KUKA KRL program: MyProgram_071().src

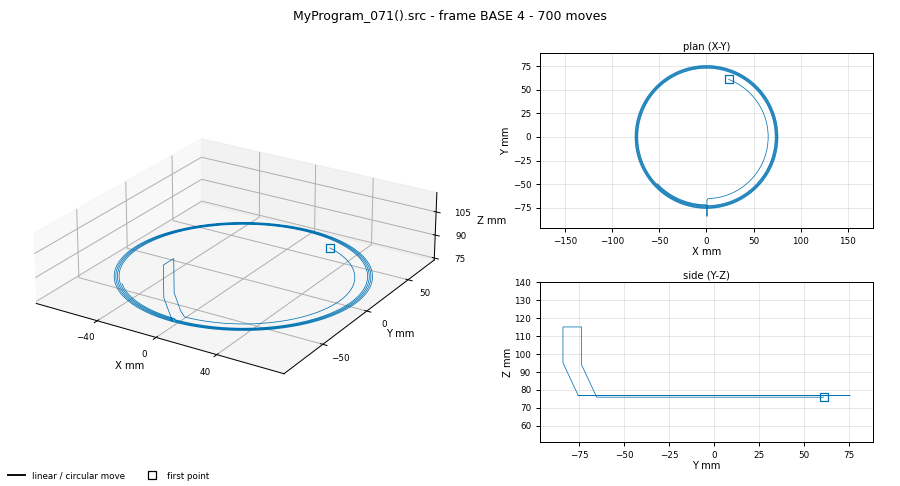
[picture p0: tool path of MyProgram_071().src in frame BASE 4, 700 of 700 moves have a stored position in this frame; points joined in program order, loops and branches not executed]
&ACCESS RVP
&REL 1
&PARAM TEMPLATE = C:\KRC\Roboter\Template\vorgabe
&PARAM EDITMASK = *
DEF MyProgram_071()
; ---- Setting reference (Base) ----
$BASE = BASE_DATA[4]

; --------------------------
; ---- Setting tool (TCP) ----
$TOOL = TOOL_DATA[3]
; --------------------------

$VEL.CP = VEL_APROX_PRINT
Startdeposition()
$VEL.CP = VEL_PRINT
LIN {X 23.5525,Y 61.0484,Z 76,A 61.9728,B 24.8705,C -2.6266,E1 25.0596,E2 22.1003} C_DIS
LIN {X 26.5205,Y 59.8189,Z 76,A 59.17,B 24.8707,C -2.6238,E1 25.0668,E2 24.903} C_DIS
LIN {X 29.4721,Y 58.4208,Z 76,A 56.3444,B 24.871,C -2.6212,E1 25.0738,E2 27.7274} C_DIS
LIN {X 32.2587,Y 56.9298,Z 76,A 53.5598,B 24.8714,C -2.617,E1 25.0807,E2 30.5137} C_DIS
LIN {X 35.0055,Y 55.2834,Z 76,A 50.8536,B 24.8716,C -2.6152,E1 25.0871,E2 33.2157} C_DIS
LIN {X 37.2904,Y 53.7671,Z 76,A 48.5544,B 24.8717,C -2.6139,E1 25.0924,E2 35.5104} C_DIS
LIN {X 39.6226,Y 52.0738,Z 76,A 45.8488,B 24.8726,C -2.6051,E1 25.0985,E2 38.2272} C_DIS
LIN {X 42.1324,Y 50.0649,Z 76,A 43.0554,B 24.873,C -2.6004,E1 25.1045,E2 41.021} C_DIS
LIN {X 44.5364,Y 47.9389,Z 76,A 40.2931,B 24.8735,C -2.596,E1 25.1102,E2 43.7826} C_DIS
LIN {X 46.2779,Y 46.26,Z 76,A 38.1504,B 24.874,C -2.591,E1 25.1145,E2 45.9282} C_DIS
LIN {X 48.4819,Y 43.9447,Z 76,A 35.3588,B 24.8745,C -2.585,E1 25.1198,E2 48.7216} C_DIS
LIN {X 50.5808,Y 41.5117,Z 76,A 32.55,B 24.8752,C -2.5787,E1 25.1249,E2 51.5324} C_DIS
LIN {X 52.564,Y 38.9698,Z 76,A 29.7557,B 24.8757,C -2.5727,E1 25.1296,E2 54.3278} C_DIS
LIN {X 54.4074,Y 36.352,Z 76,A 26.9662,B 24.8764,C -2.566,E1 25.134,E2 57.1193} C_DIS
LIN {X 55.9436,Y 33.9381,Z 76,A 24.5255,B 24.8769,C -2.5612,E1 25.1376,E2 59.559} C_DIS
LIN {X 57.326,Y 31.5494,Z 76,A 22.0724,B 24.8776,C -2.5539,E1 25.141,E2 62.0168} C_DIS
LIN {X 58.8026,Y 28.7034,Z 76,A 19.2702,B 24.8783,C -2.5463,E1 25.1445,E2 64.8219} C_DIS
LIN {X 60.1454,Y 25.7712,Z 76,A 16.4771,B 24.879,C -2.5392,E1 25.1477,E2 67.6166} C_DIS
LIN {X 61.3342,Y 22.7982,Z 76,A 13.8233,B 24.8794,C -2.5349,E1 25.1503,E2 70.2658} C_DIS
LIN {X 62.1448,Y 20.4847,Z 76,A 11.5626,B 24.8803,C -2.5257,E1 25.1524,E2 72.5355} C_DIS
LIN {X 63.0692,Y 17.4325,Z 76,A 8.7875,B 24.881,C -2.5178,E1 25.1545,E2 75.3133} C_DIS
LIN {X 63.8446,Y 14.3352,Z 76,A 6.0071,B 24.8818,C -2.5097,E1 25.1563,E2 78.0968} C_DIS
LIN {X 64.4679,Y 11.2033,Z 76,A 3.2328,B 24.8825,C -2.5017,E1 25.1577,E2 80.8738} C_DIS
LIN {X 64.9419,Y 8.0114,Z 76,A 0.4218,B 24.8833,C -2.4933,E1 25.1588,E2 83.6881} C_DIS
LIN {X 65.2564,Y 4.8203,Z 76,A -2.2442,B 24.8838,C -2.4881,E1 25.1595,E2 86.3505} C_DIS
LIN {X 65.39,Y 2.4055,Z 76,A -4.4684,B 24.8847,C -2.4787,E1 25.1597,E2 88.5837} C_DIS
LIN {X 65.4293,Y -0.8011,Z 76,A -7.1858,B 24.8853,C -2.4722,E1 25.1597,E2 91.3005} C_DIS
LIN {X 65.3532,Y -3.251,Z 76,A -9.4143,B 24.8861,C -2.4632,E1 25.1595,E2 93.5369} C_DIS
LIN {X 65.1176,Y -6.4286,Z 76,A -12.0528,B 24.8866,C -2.4583,E1 25.1588,E2 96.1713} C_DIS
LIN {X 64.8151,Y -8.9739,Z 76,A -14.3375,B 24.8873,C -2.4501,E1 25.158,E2 98.4619} C_DIS
LIN {X 64.3828,Y -11.6763,Z 76,A -16.6275,B 24.8878,C -2.4453,E1 25.157,E2 100.7497} C_DIS
LIN {X 63.8326,Y -14.3874,Z 76,A -19.1605,B 24.8887,C -2.4348,E1 25.1555,E2 103.2928} C_DIS
LIN {X 63.0604,Y -17.4644,Z 76,A -21.9235,B 24.8895,C -2.4265,E1 25.1535,E2 106.0594} C_DIS
LIN {X 62.242,Y -20.1845,Z 76,A -24.1704,B 24.8896,C -2.4251,E1 25.1516,E2 108.297} C_DIS
LIN {X 61.3315,Y -22.8052,Z 76,A -26.8132,B 24.8908,C -2.4121,E1 25.1491,E2 110.9556} C_DIS
LIN {X 60.2737,Y -25.4669,Z 76,A -29.2561,B 24.8913,C -2.4063,E1 25.1465,E2 113.3989} C_DIS
LIN {X 59.1341,Y -28.0135,Z 76,A -31.7276,B 24.8921,C -2.3983,E1 25.1436,E2 115.876} C_DIS
LIN {X 57.6977,Y -30.8641,Z 76,A -34.5052,B 24.8928,C -2.3906,E1 25.1401,E2 118.6571} C_DIS
LIN {X 56.1224,Y -33.6438,Z 76,A -37.287,B 24.8934,C -2.383,E1 25.1362,E2 121.4424} C_DIS
LIN {X 54.4127,Y -36.344,Z 76,A -40.0541,B 24.8941,C -2.376,E1 25.1319,E2 124.2122} C_DIS
LIN {X 52.4627,Y -39.1049,Z 76,A -42.9704,B 24.8947,C -2.3691,E1 25.1272,E2 127.1306} C_DIS
LIN {X 50.5595,Y -41.5372,Z 76,A -45.6811,B 24.8953,C -2.3619,E1 25.1224,E2 129.8458} C_DIS
LIN {X 48.5111,Y -43.9121,Z 76,A -48.3603,B 24.8958,C -2.3567,E1 25.1175,E2 132.5254} C_DIS
LIN {X 46.4255,Y -46.1105,Z 76,A -51.0603,B 24.8965,C -2.3491,E1 25.1122,E2 135.2318} C_DIS
LIN {X 44.1899,Y -48.2569,Z 76,A -53.7559,B 24.897,C -2.3432,E1 25.1067,E2 137.9302} C_DIS
LIN {X 41.9823,Y -50.1897,Z 76,A -56.2525,B 24.8973,C -2.3393,E1 25.1014,E2 140.4264} C_DIS
LIN {X 39.5895,Y -52.0987,Z 76,A -58.9906,B 24.898,C -2.3321,E1 25.0954,E2 143.1713} C_DIS
LIN {X 37.0025,Y -53.967,Z 76,A -61.7735,B 24.8984,C -2.3268,E1 25.089,E2 145.9571} C_DIS
LIN {X 34.3244,Y -55.7088,Z 76,A -64.5622,B 24.8989,C -2.3217,E1 25.0824,E2 148.7489} C_DIS
LIN {X 31.5458,Y -57.3279,Z 76,A -67.3726,B 24.8993,C -2.3169,E1 25.0756,E2 151.5623} C_DIS
LIN {X 28.694,Y -58.8072,Z 76,A -70.08,B 24.8995,C -2.3149,E1 25.0689,E2 154.2671} C_DIS
LIN {X 26.2021,Y -59.9577,Z 76,A -72.4647,B 24.8997,C -2.3117,E1 25.0628,E2 156.6533} C_DIS
LIN {X 23.7695,Y -60.9632,Z 76,A -74.8521,B 24.9002,C -2.3065,E1 25.0566,E2 159.0477} C_DIS
LIN {X 20.8144,Y -62.0342,Z 76,A -77.6031,B 24.9005,C -2.3031,E1 25.0493,E2 161.8014} C_DIS
LIN {X 17.8967,Y -62.938,Z 76,A -80.1335,B 24.9005,C -2.3035,E1 25.0426,E2 164.3262} C_DIS
LIN {X 15.2789,Y -63.6246,Z 76,A -82.6105,B 24.9009,C -2.2986,E1 25.0358,E2 166.8112} C_DIS
LIN {X 12.3023,Y -64.2661,Z 76,A -85.3165,B 24.9011,C -2.2954,E1 25.0284,E2 169.5215} C_DIS
LIN {X 10.0745,Y -64.6528,Z 76,A -87.1823,B 24.9011,C -2.2966,E1 25.0233,E2 171.3825} C_DIS
LIN {X 7.1628,Y -65.0407,Z 76,A -89.7299,B 24.9011,C -2.2956,E1 25.0162,E2 173.9306} C_DIS
LIN {X 4.6112,Y -65.2706,Z 76,A -91.976,B 24.9012,C -2.2945,E1 25.01,E2 176.1783} C_DIS
LIN {X 1.6014,Y -65.4146,Z 76,A -94.7265,B 24.9015,C -2.2909,E1 25.0023,E2 178.9364} C_DIS
LIN {X 1.6014,Y -65.4146,Z 76,A -94.7265,B 24.9015,C -2.2909,E1 25.0023,E2 178.9364} C_DIS
Enddeposition()
LIN {X 0.4347,Y -67.5421,Z 80.5315,A -94.7713,B 24.8999,C -2.3098,E1 25.0023,E2 178.9364} C_DIS
LIN {X 0.5123,Y -73.8809,Z 94.1262,A -94.7477,B 24.9008,C -2.2999,E1 25.0023,E2 178.9364} C_DIS
LIN {X 0.5123,Y -73.8809,Z 115.1262,A -95.1061,B 24.8873,C -2.4507,E1 25.0023,E2 178.9364} C_DIS
LIN {X 0.5071,Y -84.2101,Z 115.1262,A -95.3701,B 24.9039,C -2.2639,E1 25.0003,E2 179.6442} C_DIS
LIN {X 0.5071,Y -84.2101,Z 95.1262,A -95.0293,B 24.9157,C -2.1203,E1 25.0003,E2 179.6442} C_DIS
LIN {X 0.5079,Y -77.8709,Z 81.5315,A -95.0515,B 24.9149,C -2.1297,E1 25.0003,E2 179.6442} C_DIS
LIN {X 0.5081,Y -75.7578,Z 77,A -95.0604,B 24.9146,C -2.1334,E1 25.0003,E2 179.6442} C_DIS
Startdeposition()
$VEL.CP = VEL_PRINT
LIN {X -1.8593,Y -75.7398,Z 77,A -96.8129,B 24.9146,C -2.1341,E1 24.9954,E2 181.3953} C_DIS
LIN {X -4.4218,Y -75.6324,Z 77,A -98.7832,B 24.9146,C -2.1331,E1 24.9899,E2 183.3684} C_DIS
LIN {X -7.315,Y -75.4081,Z 77,A -100.9558,B 24.9146,C -2.1338,E1 24.9839,E2 185.5404} C_DIS
LIN {X -9.1634,Y -75.2058,Z 77,A -102.3625,B 24.9146,C -2.1339,E1 24.98,E2 186.9476} C_DIS
LIN {X -11.0062,Y -74.9583,Z 77,A -103.7692,B 24.9146,C -2.1342,E1 24.9761,E2 188.3547} C_DIS
LIN {X -12.8425,Y -74.6656,Z 77,A -105.1758,B 24.9146,C -2.1346,E1 24.9722,E2 189.7617} C_DIS
LIN {X -14.671,Y -74.328,Z 77,A -106.5836,B 24.9146,C -2.1351,E1 24.9683,E2 191.1699} C_DIS
LIN {X -16.4907,Y -73.9455,Z 77,A -107.9913,B 24.9145,C -2.1357,E1 24.9645,E2 192.5779} C_DIS
LIN {X -18.3004,Y -73.5185,Z 77,A -109.3994,B 24.9144,C -2.1364,E1 24.9607,E2 193.9863} C_DIS
LIN {X -20.0992,Y -73.0473,Z 77,A -110.8076,B 24.9144,C -2.1372,E1 24.9569,E2 195.3947} C_DIS
LIN {X -22.3492,Y -72.3898,Z 77,A -112.7026,B 24.9144,C -2.1352,E1 24.9518,E2 197.2976} C_DIS
LIN {X -24.6464,Y -71.6417,Z 77,A -114.4045,B 24.9141,C -2.1399,E1 24.9473,E2 198.9916} C_DIS
LIN {X -26.595,Y -70.9403,Z 77,A -116.1762,B 24.9144,C -2.136,E1 24.9426,E2 200.7762} C_DIS
LIN {X -28.8898,Y -70.0376,Z 77,A -117.9878,B 24.9142,C -2.1392,E1 24.9379,E2 202.5843} C_DIS
LIN {X -31.4481,Y -68.9268,Z 77,A -119.9663,B 24.9137,C -2.1448,E1 24.9329,E2 204.5541} C_DIS
LIN {X -33.8074,Y -67.8001,Z 77,A -121.9882,B 24.9137,C -2.146,E1 24.9278,E2 206.5783} C_DIS
LIN {X -35.7143,Y -66.8167,Z 77,A -123.8482,B 24.9139,C -2.142,E1 24.9232,E2 208.453} C_DIS
LIN {X -38.0527,Y -65.5124,Z 77,A -125.5985,B 24.9132,C -2.1518,E1 24.919,E2 210.1852} C_DIS
LIN {X -39.7443,Y -64.5009,Z 77,A -127.2084,B 24.9132,C -2.1509,E1 24.9151,E2 211.8022} C_DIS
LIN {X -41.9983,Y -63.0557,Z 77,A -129.1259,B 24.9128,C -2.1567,E1 24.9106,E2 213.712} C_DIS
LIN {X -43.5988,Y -61.9604,Z 77,A -130.5959,B 24.9126,C -2.159,E1 24.9073,E2 215.1815} C_DIS
LIN {X -45.1317,Y -60.8531,Z 77,A -132.0335,B 24.9124,C -2.1613,E1 24.904,E2 216.6189} C_DIS
LIN {X -46.6116,Y -59.7272,Z 77,A -133.4456,B 24.9122,C -2.1636,E1 24.9009,E2 218.0305} C_DIS
LIN {X -48.6075,Y -58.1131,Z 77,A -135.4115,B 24.912,C -2.1666,E1 24.8967,E2 219.9968} C_DIS
LIN {X -50.1864,Y -56.7565,Z 77,A -136.9756,B 24.9117,C -2.1698,E1 24.8934,E2 221.5594} C_DIS
LIN {X -51.5641,Y -55.5078,Z 77,A -138.3881,B 24.9115,C -2.1724,E1 24.8905,E2 222.9712} C_DIS
LIN {X -53.4929,Y -53.6507,Z 77,A -140.431,B 24.9112,C -2.1762,E1 24.8864,E2 225.0138} C_DIS
LIN {X -54.8709,Y -52.2414,Z 77,A -141.9205,B 24.9109,C -2.1794,E1 24.8835,E2 226.5022} C_DIS
LIN {X -56.6821,Y -50.2695,Z 77,A -143.9552,B 24.9106,C -2.1836,E1 24.8797,E2 228.5358} C_DIS
LIN {X -57.9711,Y -48.7784,Z 77,A -145.4534,B 24.9103,C -2.1868,E1 24.877,E2 230.0333} C_DIS
LIN {X -59.1507,Y -47.341,Z 77,A -147.109,B 24.9105,C -2.184,E1 24.874,E2 231.7032} C_DIS
LIN {X -60.8531,Y -45.1317,Z 77,A -148.9877,B 24.9097,C -2.1946,E1 24.8709,E2 233.5655} C_DIS
LIN {X -61.9424,Y -43.6247,Z 77,A -150.4018,B 24.9094,C -2.1979,E1 24.8686,E2 234.9788} C_DIS
LIN {X -62.9943,Y -42.0915,Z 77,A -151.8158,B 24.9091,C -2.2012,E1 24.8664,E2 236.3918} C_DIS
LIN {X -64.1223,Y -40.3503,Z 77,A -153.595,B 24.9091,C -2.2002,E1 24.8637,E2 238.1825} C_DIS
LIN {X -65.5927,Y -37.9129,Z 77,A -155.7542,B 24.9087,C -2.2057,E1 24.8606,E2 240.3398} C_DIS
LIN {X -66.9995,Y -35.3671,Z 77,A -157.8935,B 24.9081,C -2.213,E1 24.8578,E2 242.4728} C_DIS
LIN {X -68.0859,Y -33.2307,Z 77,A -159.8507,B 24.9081,C -2.2145,E1 24.8554,E2 244.437} C_DIS
LIN {X -69.2629,Y -30.7021,Z 77,A -161.7188,B 24.907,C -2.2262,E1 24.8532,E2 246.2875} C_DIS
LIN {X -69.9955,Y -28.9931,Z 77,A -163.1343,B 24.9067,C -2.2299,E1 24.8517,E2 247.7019} C_DIS
LIN {X -70.686,Y -27.2666,Z 77,A -164.5499,B 24.9064,C -2.2338,E1 24.8502,E2 249.1163} C_DIS
LIN {X -71.3338,Y -25.5237,Z 77,A -165.9652,B 24.9061,C -2.2376,E1 24.8489,E2 250.5303} C_DIS
LIN {X -71.9031,Y -23.8711,Z 77,A -167.3043,B 24.9058,C -2.2411,E1 24.8477,E2 251.8687} C_DIS
LIN {X -72.733,Y -21.2083,Z 77,A -169.4276,B 24.9053,C -2.2471,E1 24.846,E2 253.99} C_DIS
LIN {X -73.4125,Y -18.7184,Z 77,A -171.4427,B 24.9049,C -2.2514,E1 24.8445,E2 256.0064} C_DIS
LIN {X -73.9744,Y -16.3584,Z 77,A -173.4176,B 24.9047,C -2.2537,E1 24.8433,E2 257.9874} C_DIS
LIN {X -74.4826,Y -13.8676,Z 77,A -175.2484,B 24.904,C -2.2618,E1 24.8423,E2 259.8099} C_DIS
LIN {X -74.9256,Y -11.2269,Z 77,A -177.2155,B 24.9034,C -2.2694,E1 24.8414,E2 261.7704} C_DIS
LIN {X -75.246,Y -8.8201,Z 77,A -179.1504,B 24.9031,C -2.2728,E1 24.8407,E2 263.7087} C_DIS
LIN {X -75.4833,Y -6.5002,Z 77,A 179.168,B 24.9024,C -2.2803,E1 24.8403,E2 265.3827} C_DIS
LIN {X -75.6652,Y -3.8289,Z 77,A 177.1202,B 24.9019,C -2.2861,E1 24.8399,E2 267.4288} C_DIS
LIN {X -75.7549,Y -1.0413,Z 77,A 174.7529,B 24.9019,C -2.2868,E1 24.8398,E2 269.8088} C_DIS
LIN {X -75.7398,Y 1.8593,Z 77,A 172.7949,B 24.9008,C -2.2992,E1 24.8398,E2 271.7488} C_DIS
LIN {X -75.6761,Y 3.606,Z 77,A 171.3838,B 24.9006,C -2.3014,E1 24.84,E2 273.1633} C_DIS
LIN {X -75.4937,Y 6.3697,Z 77,A 169.3521,B 24.8999,C -2.3095,E1 24.8404,E2 275.1878} C_DIS
LIN {X -75.301,Y 8.3507,Z 77,A 167.8383,B 24.8995,C -2.3141,E1 24.8409,E2 276.6998} C_DIS
LIN {X -75.0734,Y 10.1962,Z 77,A 166.4219,B 24.8992,C -2.3183,E1 24.8414,E2 278.1146} C_DIS
LIN {X -74.7112,Y 12.5698,Z 77,A 164.3699,B 24.8992,C -2.3185,E1 24.8423,E2 280.1781} C_DIS
LIN {X -74.1199,Y 15.6913,Z 77,A 162.1728,B 24.8981,C -2.3309,E1 24.8435,E2 282.3588} C_DIS
LIN {X -73.7125,Y 17.5056,Z 77,A 160.7567,B 24.8977,C -2.3351,E1 24.8444,E2 283.7732} C_DIS
LIN {X -73.2607,Y 19.3093,Z 77,A 159.3407,B 24.8973,C -2.3392,E1 24.8453,E2 285.1875} C_DIS
LIN {X -72.7647,Y 21.1014,Z 77,A 157.9247,B 24.897,C -2.3434,E1 24.8464,E2 286.6018} C_DIS
LIN {X -72.225,Y 22.8808,Z 77,A 156.5087,B 24.8966,C -2.3475,E1 24.8476,E2 288.0161} C_DIS
LIN {X -71.6417,Y 24.6464,Z 77,A 154.8804,B 24.8966,C -2.3466,E1 24.8491,E2 289.6558} C_DIS
LIN {X -70.7255,Y 27.1623,Z 77,A 153.045,B 24.8957,C -2.3572,E1 24.8508,E2 291.4763} C_DIS
LIN {X -69.7451,Y 29.5874,Z 77,A 151.0139,B 24.8953,C -2.3619,E1 24.853,E2 293.5074} C_DIS
LIN {X -68.9268,Y 31.4481,Z 77,A 149.3728,B 24.8951,C -2.3641,E1 24.8549,E2 295.1524} C_DIS
LIN {X -67.7226,Y 33.9638,Z 77,A 147.3824,B 24.8943,C -2.3731,E1 24.8573,E2 297.1321} C_DIS
LIN {X -66.8686,Y 35.6155,Z 77,A 145.967,B 24.894,C -2.3769,E1 24.8591,E2 298.5458} C_DIS
LIN {X -65.7568,Y 37.6275,Z 77,A 144.0566,B 24.8939,C -2.3779,E1 24.8617,E2 300.464} C_DIS
LIN {X -64.5009,Y 39.7443,Z 77,A 142.3527,B 24.8931,C -2.3868,E1 24.8642,E2 302.1553} C_DIS
LIN {X -62.9943,Y 42.0915,Z 77,A 140.23,B 24.8926,C -2.3923,E1 24.8674,E2 304.2755} C_DIS
LIN {X -61.6349,Y 44.0557,Z 77,A 138.1767,B 24.8926,C -2.3914,E1 24.8707,E2 306.3411} C_DIS
LIN {X -59.7272,Y 46.6116,Z 77,A 135.9861,B 24.8916,C -2.403,E1 24.8744,E2 308.5144} C_DIS
LIN {X -58.0424,Y 48.6926,Z 77,A 133.9493,B 24.8912,C -2.408,E1 24.878,E2 310.5489} C_DIS
LIN {X -56.8299,Y 50.1023,Z 77,A 132.5264,B 24.8909,C -2.4111,E1 24.8806,E2 311.9707} C_DIS
LIN {X -55.5078,Y 51.5641,Z 77,A 130.7939,B 24.8911,C -2.409,E1 24.8839,E2 313.7159} C_DIS
LIN {X -53.5723,Y 53.5723,Z 77,A 128.6328,B 24.8907,C -2.4128,E1 24.8881,E2 315.8771} C_DIS
LIN {X -51.3931,Y 55.6647,Z 77,A 126.4255,B 24.8901,C -2.42,E1 24.8926,E2 318.0763} C_DIS
LIN {X -49.5701,Y 57.2947,Z 77,A 124.7509,B 24.8893,C -2.4283,E1 24.8961,E2 319.7376} C_DIS
LIN {X -47.4277,Y 59.0805,Z 77,A 122.4512,B 24.8893,C -2.4283,E1 24.9011,E2 322.0462} C_DIS
LIN {X -45.1317,Y 60.8531,Z 77,A 120.4362,B 24.8885,C -2.4372,E1 24.9055,E2 324.0472} C_DIS
LIN {X -43.6247,Y 61.9424,Z 77,A 119.0235,B 24.8883,C -2.4398,E1 24.9087,E2 325.4585} C_DIS
LIN {X -42.0915,Y 62.9943,Z 77,A 117.611,B 24.888,C -2.4424,E1 24.912,E2 326.8696} C_DIS
LIN {X -40.6267,Y 63.9481,Z 77,A 116.0362,B 24.8884,C -2.4387,E1 24.9157,E2 328.4583} C_DIS
LIN {X -38.1494,Y 65.4568,Z 77,A 114.0099,B 24.8876,C -2.4467,E1 24.9206,E2 330.4716} C_DIS
LIN {X -35.8471,Y 66.7446,Z 77,A 112.074,B 24.8872,C -2.4516,E1 24.9253,E2 332.4015} C_DIS
LIN {X -34.1631,Y 67.6222,Z 77,A 110.6284,B 24.887,C -2.4537,E1 24.9289,E2 333.846} C_DIS
LIN {X -32.4932,Y 68.4403,Z 77,A 109.0424,B 24.8872,C -2.4514,E1 24.9329,E2 335.4415} C_DIS
LIN {X -29.9521,Y 69.5899,Z 77,A 107.101,B 24.8865,C -2.4587,E1 24.9378,E2 337.3703} C_DIS
LIN {X -28.132,Y 70.3461,Z 77,A 105.614,B 24.8863,C -2.4608,E1 24.9416,E2 338.8555} C_DIS
LIN {X -26.3971,Y 71.0153,Z 77,A 103.9456,B 24.8868,C -2.456,E1 24.946,E2 340.5387} C_DIS
LIN {X -23.8711,Y 71.9031,Z 77,A 102.1647,B 24.886,C -2.4647,E1 24.9507,E2 342.3025} C_DIS
LIN {X -21.2083,Y 72.733,Z 77,A 100.0588,B 24.8858,C -2.4671,E1 24.9563,E2 344.4062} C_DIS
LIN {X -19.3093,Y 73.2607,Z 77,A 98.565,B 24.8856,C -2.4685,E1 24.9603,E2 345.899} C_DIS
LIN {X -17.5056,Y 73.7125,Z 77,A 97.1554,B 24.8856,C -2.4697,E1 24.9642,E2 347.3076} C_DIS
LIN {X -15.6913,Y 74.1199,Z 77,A 95.4735,B 24.8861,C -2.4639,E1 24.9688,E2 349.0054} C_DIS
LIN {X -13.0623,Y 74.6275,Z 77,A 93.7096,B 24.8853,C -2.4722,E1 24.9736,E2 350.7516} C_DIS
LIN {X -10.8615,Y 74.9789,Z 77,A 91.8499,B 24.8856,C -2.4688,E1 24.9788,E2 352.6208} C_DIS
LIN {X -8.3507,Y 75.301,Z 77,A 89.909,B 24.8856,C -2.4692,E1 24.9841,E2 354.5621} C_DIS
LIN {X -5.5734,Y 75.5573,Z 77,A 88.0013,B 24.885,C -2.4754,E1 24.9894,E2 356.456} C_DIS
LIN {X -2.9846,Y 75.7029,Z 77,A 86.0273,B 24.885,C -2.4758,E1 24.9949,E2 358.4296} C_DIS
LIN {X -1.0663,Y 75.7544,Z 77,A 84.3242,B 24.8855,C -2.4695,E1 24.9997,E2 360.1476} C_DIS
LIN {X 1.8593,Y 75.7398,Z 77,A 82.3732,B 24.8849,C -2.4767,E1 25.0051,E2 362.0813} C_DIS
LIN {X 3.606,Y 75.6761,Z 77,A 81.0424,B 24.8849,C -2.4766,E1 25.0088,E2 363.412} C_DIS
LIN {X 5.5734,Y 75.5573,Z 77,A 79.5609,B 24.8849,C -2.4768,E1 25.0129,E2 364.8924} C_DIS
LIN {X 8.3507,Y 75.301,Z 77,A 77.4522,B 24.8849,C -2.4766,E1 25.0188,E2 367.0003} C_DIS
LIN {X 10.4168,Y 75.042,Z 77,A 75.6607,B 24.8855,C -2.4704,E1 25.0238,E2 368.8049} C_DIS
LIN {X 12.8425,Y 74.6656,Z 77,A 74.0143,B 24.885,C -2.4755,E1 25.0283,E2 370.4376} C_DIS
LIN {X 14.671,Y 74.328,Z 77,A 72.6093,B 24.885,C -2.4749,E1 25.0322,E2 371.8423} C_DIS
LIN {X 17.2224,Y 73.7779,Z 77,A 70.6125,B 24.8852,C -2.4733,E1 25.0376,E2 373.8403} C_DIS
LIN {X 19.2371,Y 73.2792,Z 77,A 69.0808,B 24.8852,C -2.4734,E1 25.0417,E2 375.3695} C_DIS
LIN {X 21.1014,Y 72.7647,Z 77,A 67.5473,B 24.8854,C -2.4705,E1 25.0459,E2 376.9073} C_DIS
LIN {X 23.6061,Y 71.9903,Z 77,A 65.6202,B 24.8854,C -2.4705,E1 25.051,E2 378.8309} C_DIS
LIN {X 25.4184,Y 71.3708,Z 77,A 64.1842,B 24.8855,C -2.4696,E1 25.0548,E2 380.2662} C_DIS
LIN {X 27.2297,Y 70.6999,Z 77,A 62.7376,B 24.8856,C -2.4686,E1 25.0586,E2 381.712} C_DIS
LIN {X 28.8898,Y 70.0376,Z 77,A 61.378,B 24.8858,C -2.467,E1 25.0621,E2 383.0723} C_DIS
LIN {X 30.6872,Y 69.2694,Z 77,A 59.9134,B 24.8858,C -2.4658,E1 25.0658,E2 384.5362} C_DIS
LIN {X 32.3927,Y 68.4886,Z 77,A 58.497,B 24.886,C -2.4642,E1 25.0694,E2 385.9528} C_DIS
LIN {X 34.5281,Y 67.4357,Z 77,A 56.6311,B 24.8864,C -2.4602,E1 25.0741,E2 387.8232} C_DIS
LIN {X 36.5315,Y 66.3734,Z 77,A 54.7344,B 24.8871,C -2.4528,E1 25.0788,E2 389.732} C_DIS
LIN {X 38.8537,Y 65.0405,Z 77,A 52.9638,B 24.8867,C -2.457,E1 25.083,E2 391.4871} C_DIS
LIN {X 41.2163,Y 63.5696,Z 77,A 50.8746,B 24.887,C -2.4542,E1 25.0879,E2 393.5762} C_DIS
LIN {X 42.769,Y 62.5356,Z 77,A 49.4693,B 24.8871,C -2.4521,E1 25.0912,E2 394.9818} C_DIS
LIN {X 44.2908,Y 61.4672,Z 77,A 48.0597,B 24.8874,C -2.4497,E1 25.0944,E2 396.3923} C_DIS
LIN {X 45.8751,Y 60.2947,Z 77,A 46.5836,B 24.8876,C -2.4475,E1 25.0977,E2 397.8683} C_DIS
LIN {X 47.341,Y 59.1507,Z 77,A 45.183,B 24.8878,C -2.4451,E1 25.1008,E2 399.2693} C_DIS
LIN {X 49.3944,Y 57.4462,Z 77,A 43.1632,B 24.8882,C -2.4412,E1 25.1051,E2 401.2904} C_DIS
LIN {X 50.796,Y 56.2108,Z 77,A 41.7578,B 24.8884,C -2.4387,E1 25.108,E2 402.6963} C_DIS
LIN {X 52.2414,Y 54.8709,Z 77,A 40.2824,B 24.8886,C -2.4361,E1 25.111,E2 404.1718} C_DIS
LIN {X 53.4929,Y 53.6507,Z 77,A 38.9583,B 24.8889,C -2.4332,E1 25.1137,E2 405.497} C_DIS
LIN {X 54.7934,Y 52.3217,Z 77,A 37.5588,B 24.8891,C -2.4304,E1 25.1164,E2 406.8971} C_DIS
LIN {X 56.1364,Y 50.8791,Z 77,A 36.0839,B 24.8894,C -2.4276,E1 25.1192,E2 408.3723} C_DIS
LIN {X 57.3681,Y 49.4861,Z 77,A 34.6847,B 24.8897,C -2.4246,E1 25.1217,E2 409.7722} C_DIS
LIN {X 58.5653,Y 48.0633,Z 77,A 33.2856,B 24.89,C -2.4216,E1 25.1242,E2 411.1721} C_DIS
LIN {X 59.7272,Y 46.6116,Z 77,A 31.8867,B 24.8902,C -2.4185,E1 25.1267,E2 412.5718} C_DIS
LIN {X 60.8531,Y 45.1317,Z 77,A 30.4882,B 24.8905,C -2.4153,E1 25.129,E2 413.9712} C_DIS
LIN {X 61.8776,Y 43.7155,Z 77,A 29.0846,B 24.891,C -2.4096,E1 25.1313,E2 415.3813} C_DIS
LIN {X 63.4447,Y 41.4084,Z 77,A 27.0673,B 24.8913,C -2.407,E1 25.1344,E2 417.3947} C_DIS
LIN {X 64.7248,Y 39.3758,Z 77,A 25.1661,B 24.8919,C -2.3998,E1 25.1372,E2 419.3033} C_DIS
LIN {X 65.8645,Y 37.44,Z 77,A 23.3912,B 24.8925,C -2.3931,E1 25.1397,E2 421.0849} C_DIS
LIN {X 67.2499,Y 34.8916,Z 77,A 21.4001,B 24.8925,C -2.3931,E1 25.1423,E2 423.0655} C_DIS
LIN {X 68.0859,Y 33.2307,Z 77,A 19.8587,B 24.8932,C -2.3852,E1 25.1442,E2 424.6174} C_DIS
LIN {X 69.2629,Y 30.7021,Z 77,A 17.9065,B 24.8934,C -2.384,E1 25.1465,E2 426.5619} C_DIS
LIN {X 70.3461,Y 28.132,Z 77,A 15.8104,B 24.8939,C -2.3783,E1 25.1487,E2 428.6598} C_DIS
LIN {X 71.0153,Y 26.3971,Z 77,A 14.3101,B 24.8945,C -2.3714,E1 25.1502,E2 430.168} C_DIS
LIN {X 71.9031,Y 23.8711,Z 77,A 12.3926,B 24.8947,C -2.3687,E1 25.152,E2 432.0811} C_DIS
LIN {X 72.6863,Y 21.3657,Z 77,A 10.4001,B 24.8953,C -2.3626,E1 25.1536,E2 434.0768} C_DIS
LIN {X 73.3862,Y 18.8207,Z 77,A 8.352,B 24.8959,C -2.355,E1 25.1551,E2 436.131} C_DIS
LIN {X 73.8966,Y 16.7084,Z 77,A 6.8055,B 24.8961,C -2.3529,E1 25.1561,E2 437.6735} C_DIS
LIN {X 74.2844,Y 14.8898,Z 77,A 5.4085,B 24.8965,C -2.3489,E1 25.1569,E2 439.0719} C_DIS
LIN {X 74.6275,Y 13.0623,Z 77,A 4.0121,B 24.8968,C -2.3448,E1 25.1576,E2 440.4697} C_DIS
LIN {X 74.9256,Y 11.2269,Z 77,A 2.6152,B 24.8972,C -2.3407,E1 25.1582,E2 441.868} C_DIS
LIN {X 75.2164,Y 9.0727,Z 77,A 0.787,B 24.8981,C -2.3301,E1 25.1588,E2 443.7106} C_DIS
LIN {X 75.4833,Y 6.5002,Z 77,A -0.9511,B 24.8981,C -2.3304,E1 25.1593,E2 445.4376} C_DIS
LIN {X 75.6125,Y 4.7571,Z 77,A -2.4438,B 24.8989,C -2.3211,E1 25.1596,E2 446.9434} C_DIS
LIN {X 75.7364,Y 1.9708,Z 77,A -4.3494,B 24.8989,C -2.3206,E1 25.1597,E2 448.8389} C_DIS
LIN {X 75.762,Y 0,Z 77,A -5.8793,B 24.8995,C -2.3146,E1 25.1597,E2 450.3737} C_DIS
LIN {X 75.7113,Y -2.7886,Z 77,A -7.9327,B 24.8999,C -2.3096,E1 25.1597,E2 452.4268} C_DIS
LIN {X 75.62,Y -4.6458,Z 77,A -9.3288,B 24.9003,C -2.3054,E1 25.1594,E2 453.8245} C_DIS
LIN {X 75.4081,Y -7.315,Z 77,A -11.3485,B 24.9008,C -2.2991,E1 25.1589,E2 455.847} C_DIS
LIN {X 75.2058,Y -9.1634,Z 77,A -12.7448,B 24.9012,C -2.295,E1 25.1585,E2 457.245} C_DIS
LIN {X 74.9583,Y -11.0062,Z 77,A -14.2796,B 24.9019,C -2.2866,E1 25.1579,E2 458.7904} C_DIS
LIN {X 74.4826,Y -13.8676,Z 77,A -16.3107,B 24.9021,C -2.2846,E1 25.1569,E2 460.8145} C_DIS
LIN {X 74.1199,Y -15.6913,Z 77,A -17.7073,B 24.9024,C -2.2804,E1 25.1561,E2 462.2128} C_DIS
LIN {X 73.7125,Y -17.5056,Z 77,A -19.1036,B 24.9028,C -2.2763,E1 25.1553,E2 463.6107} C_DIS
LIN {X 73.2607,Y -19.3093,Z 77,A -20.5,B 24.9031,C -2.2722,E1 25.1543,E2 465.0088} C_DIS
LIN {X 72.5074,Y -21.9688,Z 77,A -22.5766,B 24.9037,C -2.2661,E1 25.1527,E2 467.0878} C_DIS
LIN {X 71.9731,Y -23.6592,Z 77,A -23.9163,B 24.904,C -2.262,E1 25.1515,E2 468.4297} C_DIS
LIN {X 71.0535,Y -26.2923,Z 77,A -26.0111,B 24.9045,C -2.2559,E1 25.1496,E2 470.527} C_DIS
LIN {X 70.3868,Y -28.0281,Z 77,A -27.5734,B 24.9053,C -2.247,E1 25.148,E2 472.1017} C_DIS
LIN {X 69.2629,Y -30.7021,Z 77,A -29.5783,B 24.9053,C -2.246,E1 25.1458,E2 474.098} C_DIS
LIN {X 68.4886,Y -32.3927,Z 77,A -30.9754,B 24.9057,C -2.2421,E1 25.1441,E2 475.4968} C_DIS
LIN {X 67.7226,Y -33.9638,Z 77,A -32.2972,B 24.906,C -2.2382,E1 25.1425,E2 476.8207} C_DIS
LIN {X 66.8167,Y -35.7143,Z 77,A -33.9792,B 24.9069,C -2.2281,E1 25.1403,E2 478.5176} C_DIS
LIN {X 65.5386,Y -38.0072,Z 77,A -35.7485,B 24.9069,C -2.2289,E1 25.1378,E2 480.276} C_DIS
LIN {X 64.5009,Y -39.7443,Z 77,A -37.263,B 24.9071,C -2.225,E1 25.1356,E2 481.7919} C_DIS
LIN {X 63.2778,Y -41.6615,Z 77,A -39.102,B 24.9078,C -2.2167,E1 25.1328,E2 483.6414} C_DIS
LIN {X 61.5922,Y -44.1154,Z 77,A -41.2704,B 24.9081,C -2.213,E1 25.1294,E2 485.8079} C_DIS
LIN {X 60.3617,Y -45.7859,Z 77,A -42.7786,B 24.9083,C -2.2106,E1 25.1269,E2 487.3146} C_DIS
LIN {X 59.2199,Y -47.2535,Z 77,A -44.4121,B 24.9092,C -2.2001,E1 25.124,E2 488.965} C_DIS
LIN {X 57.4405,Y -49.4012,Z 77,A -46.274,B 24.909,C -2.202,E1 25.1207,E2 490.814} C_DIS
LIN {X 55.9104,Y -51.1253,Z 77,A -48.143,B 24.9097,C -2.1939,E1 25.1172,E2 492.6938} C_DIS
LIN {X 54.3031,Y -52.8305,Z 77,A -49.7618,B 24.9097,C -2.1941,E1 25.114,E2 494.3052} C_DIS
LIN {X 52.9108,Y -54.2256,Z 77,A -51.2441,B 24.91,C -2.1907,E1 25.1111,E2 495.7892} C_DIS
LIN {X 51.5641,Y -55.5078,Z 77,A -52.643,B 24.9102,C -2.1876,E1 25.1083,E2 497.1896} C_DIS
LIN {X 49.4861,Y -57.3681,Z 77,A -55.0258,B 24.9113,C -2.1748,E1 25.1032,E2 499.5933} C_DIS
LIN {X 47.341,Y -59.1507,Z 77,A -56.8408,B 24.911,C -2.1788,E1 25.0993,E2 501.392} C_DIS
LIN {X 45.5749,Y -60.5202,Z 77,A -58.6497,B 24.9115,C -2.1718,E1 25.0953,E2 503.2108} C_DIS
LIN {X 43.6988,Y -61.8895,Z 77,A -60.2704,B 24.9115,C -2.1722,E1 25.0916,E2 504.825} C_DIS
LIN {X 42.0915,Y -62.9943,Z 77,A -61.7403,B 24.9117,C -2.1694,E1 25.0882,E2 506.2965} C_DIS
LIN {X 40.6267,Y -63.9481,Z 77,A -63.0653,B 24.9119,C -2.1668,E1 25.0851,E2 507.6234} C_DIS
LIN {X 39.0451,Y -64.9258,Z 77,A -64.4659,B 24.9121,C -2.1643,E1 25.0818,E2 509.0254} C_DIS
LIN {X 37.1159,Y -66.047,Z 77,A -66.3156,B 24.9128,C -2.1567,E1 25.0773,E2 510.8877} C_DIS
LIN {X 34.5646,Y -67.4171,Z 77,A -68.4702,B 24.913,C -2.154,E1 25.0719,E2 513.0426} C_DIS
LIN {X 31.6509,Y -68.8339,Z 77,A -70.7703,B 24.913,C -2.1544,E1 25.0662,E2 515.3356} C_DIS
LIN {X 29.9521,Y -69.5899,Z 77,A -72.3302,B 24.9135,C -2.148,E1 25.0621,E2 516.9071} C_DIS
LIN {X 27.2666,Y -70.686,Z 77,A -74.3506,B 24.9133,C -2.1498,E1 25.0569,E2 518.9186} C_DIS
LIN {X 25.5237,Y -71.3338,Z 77,A -75.7526,B 24.9135,C -2.1481,E1 25.0532,E2 520.3217} C_DIS
LIN {X 23.8711,Y -71.9031,Z 77,A -77.0792,B 24.9135,C -2.1463,E1 25.0497,E2 521.6499} C_DIS
LIN {X 21.7534,Y -72.5713,Z 77,A -78.9286,B 24.9141,C -2.1396,E1 25.0448,E2 523.5119} C_DIS
LIN {X 19.3093,Y -73.2607,Z 77,A -80.6615,B 24.9139,C -2.1428,E1 25.0401,E2 525.2344} C_DIS
LIN {X 17.5056,Y -73.7125,Z 77,A -82.0651,B 24.9139,C -2.1415,E1 25.0363,E2 526.639} C_DIS
LIN {X 15.6913,Y -74.1199,Z 77,A -83.4683,B 24.9141,C -2.1403,E1 25.0325,E2 528.0433} C_DIS
LIN {X 13.8676,Y -74.4826,Z 77,A -84.8721,B 24.9141,C -2.1392,E1 25.0286,E2 529.448} C_DIS
LIN {X 11.4882,Y -74.8852,Z 77,A -86.7711,B 24.9144,C -2.1359,E1 25.0234,E2 531.3531} C_DIS
LIN {X 9.3848,Y -75.1785,Z 77,A -88.3067,B 24.9144,C -2.1368,E1 25.0191,E2 532.8853} C_DIS
LIN {X 7.537,Y -75.3862,Z 77,A -89.8181,B 24.9147,C -2.1331,E1 25.0149,E2 534.4044} C_DIS
LIN {X 4.7571,Y -75.6125,Z 77,A -91.8093,B 24.9145,C -2.1353,E1 25.0094,E2 536.3893} C_DIS
LIN {X 2.7886,Y -75.7113,Z 77,A -93.299,B 24.9145,C -2.1348,E1 25.0052,E2 537.8799} C_DIS
LIN {X 0.5081,Y -75.7578,Z 77,A -95.06,B 24.9146,C -2.1334,E1 25.0003,E2 539.6439} C_DIS
Enddeposition()
LIN {X 0.5081,Y -75.7578,Z 77,A -95.06,B 24.9146,C -2.1334,E1 25.0003,E2 539.6439} C_DIS
Startdeposition()
$VEL.CP = VEL_PRINT
LIN {X 1.7839,Y -74.7888,Z 77,A -93.4248,B 24.9118,C -2.1681,E1 25.0051,E2 537.9266} C_DIS
LIN {X 3.8573,Y -74.71,Z 77,A -91.6001,B 24.9113,C -2.1751,E1 25.0102,E2 536.0858} C_DIS
LIN {X 6.817,Y -74.4977,Z 77,A -89.4436,B 24.9114,C -2.1731,E1 25.0162,E2 533.9353} C_DIS
LIN {X 9.6182,Y -74.1881,Z 77,A -87.142,B 24.911,C -2.1783,E1 25.0226,E2 531.6229} C_DIS
LIN {X 13.3654,Y -73.6055,Z 77,A -83.9112,B 24.9101,C -2.1896,E1 25.0316,E2 528.3686} C_DIS
LIN {X 19.3223,Y -72.2708,Z 77,A -79.7087,B 24.9108,C -2.1808,E1 25.0429,E2 524.1931} C_DIS
LIN {X 22.5597,Y -71.3274,Z 77,A -77.3106,B 24.911,C -2.1785,E1 25.0493,E2 521.8046} C_DIS
LIN {X 25.8085,Y -70.2164,Z 77,A -74.3793,B 24.91,C -2.1904,E1 25.0571,E2 518.8511} C_DIS
LIN {X 28.5127,Y -69.163,Z 77,A -71.5677,B 24.9083,C -2.2104,E1 25.0645,E2 515.9985} C_DIS
LIN {X 31.5067,Y -67.8507,Z 77,A -69.1583,B 24.9083,C -2.2116,E1 25.0706,E2 513.5925} C_DIS
LIN {X 35.1012,Y -66.0633,Z 77,A -66.6053,B 24.9091,C -2.2016,E1 25.0768,E2 511.0703} C_DIS
LIN {X 39.7481,Y -63.3758,Z 77,A -62.7439,B 24.9091,C -2.2018,E1 25.0861,E2 507.2202} C_DIS
LIN {X 41.7034,Y -62.1071,Z 77,A -60.7633,B 24.9083,C -2.2109,E1 25.0907,E2 505.2245} C_DIS
LIN {X 44.2439,Y -60.323,Z 77,A -58.422,B 24.908,C -2.2147,E1 25.096,E2 502.8825} C_DIS
LIN {X 46.6571,Y -58.4775,Z 77,A -55.7953,B 24.9068,C -2.2285,E1 25.1018,E2 500.2329} C_DIS
LIN {X 49.7013,Y -55.9127,Z 77,A -53.4132,B 24.9079,C -2.2158,E1 25.1068,E2 497.8902} C_DIS
LIN {X 51.1621,Y -54.5787,Z 77,A -51.5094,B 24.9067,C -2.2307,E1 25.1108,E2 495.9589} C_DIS
LIN {X 53.2696,Y -52.5236,Z 77,A -49.2815,B 24.9063,C -2.2353,E1 25.1152,E2 493.7295} C_DIS
LIN {X 55.7335,Y -49.9015,Z 77,A -46.2363,B 24.905,C -2.2508,E1 25.121,E2 490.661} C_DIS
LIN {X 57.7126,Y -47.5996,Z 77,A -44.3121,B 24.9055,C -2.2449,E1 25.1244,E2 488.7598} C_DIS
LIN {X 59.5558,Y -45.2733,Z 77,A -41.9722,B 24.9048,C -2.2529,E1 25.1284,E2 486.4119} C_DIS
LIN {X 61.3138,Y -42.8606,Z 77,A -39.7469,B 24.9044,C -2.2573,E1 25.132,E2 484.1871} C_DIS
LIN {X 62.9119,Y -40.4781,Z 77,A -36.6857,B 24.9017,C -2.2894,E1 25.1367,E2 481.0653} C_DIS
LIN {X 64.9411,Y -37.1358,Z 77,A -34.4834,B 24.903,C -2.2741,E1 25.1397,E2 478.9107} C_DIS
LIN {X 66.422,Y -34.4191,Z 77,A -32.1697,B 24.9025,C -2.2793,E1 25.1428,E2 476.5969} C_DIS
LIN {X 67.7705,Y -31.6789,Z 77,A -29.8807,B 24.9021,C -2.2847,E1 25.1455,E2 474.3073} C_DIS
LIN {X 68.9306,Y -29.0682,Z 77,A -27.6743,B 24.9015,C -2.2918,E1 25.148,E2 472.0962} C_DIS
LIN {X 70.1068,Y -26.1058,Z 77,A -25.3127,B 24.901,C -2.2969,E1 25.1503,E2 469.7358} C_DIS
LIN {X 71.0944,Y -23.2813,Z 77,A -22.8934,B 24.9001,C -2.3078,E1 25.1525,E2 467.3043} C_DIS
LIN {X 71.8802,Y -20.7301,Z 77,A -21.0528,B 24.9001,C -2.308,E1 25.1539,E2 465.4739} C_DIS
LIN {X 72.6091,Y -18.0106,Z 77,A -18.8987,B 24.8995,C -2.3147,E1 25.1555,E2 463.3163} C_DIS
LIN {X 73.215,Y -15.3642,Z 77,A -16.7949,B 24.8988,C -2.3219,E1 25.1567,E2 461.2076} C_DIS
LIN {X 73.734,Y -12.6401,Z 77,A -14.698,B 24.8983,C -2.3279,E1 25.1578,E2 459.109} C_DIS
LIN {X 74.1481,Y -9.9268,Z 77,A -12.6018,B 24.8978,C -2.3344,E1 25.1586,E2 457.0098} C_DIS
LIN {X 74.497,Y -6.8254,Z 77,A -10.5716,B 24.898,C -2.3311,E1 25.1592,E2 454.9993} C_DIS
LIN {X 74.6451,Y -4.9502,Z 77,A -8.6466,B 24.8963,C -2.3503,E1 25.1596,E2 453.0403} C_DIS
LIN {X 74.7676,Y -2.496,Z 77,A -6.9604,B 24.8963,C -2.3503,E1 25.1597,E2 451.364} C_DIS
LIN {X 74.806,Y 0.7123,Z 77,A -4.3652,B 24.8953,C -2.3624,E1 25.1597,E2 448.7559} C_DIS
LIN {X 74.6984,Y 4.0665,Z 77,A -2.0294,B 24.8952,C -2.3634,E1 25.1595,E2 446.4315} C_DIS
LIN {X 74.5012,Y 6.7795,Z 77,A 0.0564,B 24.8946,C -2.3701,E1 25.159,E2 444.3424} C_DIS
LIN {X 74.2265,Y 9.3218,Z 77,A 2.0732,B 24.8939,C -2.3779,E1 25.1583,E2 442.319} C_DIS
LIN {X 73.8364,Y 12.0277,Z 77,A 4.1824,B 24.8933,C -2.3849,E1 25.1574,E2 440.2057} C_DIS
LIN {X 73.2184,Y 15.3476,Z 77,A 6.6635,B 24.8928,C -2.3897,E1 25.1561,E2 437.7278} C_DIS
LIN {X 72.541,Y 18.2839,Z 77,A 9.0785,B 24.8919,C -2.3999,E1 25.1545,E2 435.3025} C_DIS
LIN {X 71.6537,Y 21.4985,Z 77,A 11.6266,B 24.8912,C -2.4074,E1 25.1525,E2 432.7514} C_DIS
LIN {X 70.436,Y 25.2063,Z 77,A 14.6157,B 24.8904,C -2.4162,E1 25.1498,E2 429.7585} C_DIS
LIN {X 69.2909,Y 28.1984,Z 77,A 16.9393,B 24.8902,C -2.4194,E1 25.1475,E2 427.4401} C_DIS
LIN {X 68.2634,Y 30.6025,Z 77,A 18.922,B 24.8897,C -2.4244,E1 25.1452,E2 425.4562} C_DIS
LIN {X 67.0041,Y 33.2691,Z 77,A 21.1477,B 24.8892,C -2.4297,E1 25.1425,E2 423.2301} C_DIS
LIN {X 65.708,Y 35.7611,Z 77,A 23.8903,B 24.8871,C -2.4531,E1 25.1388,E2 420.4466} C_DIS
LIN {X 63.742,Y 39.1595,Z 77,A 26.2437,B 24.8881,C -2.4416,E1 25.1355,E2 418.1324} C_DIS
LIN {X 62.2422,Y 41.5024,Z 77,A 28.5216,B 24.8872,C -2.4513,E1 25.132,E2 415.8428} C_DIS
LIN {X 59.928,Y 44.7778,Z 77,A 31.4071,B 24.887,C -2.4534,E1 25.1273,E2 412.9664} C_DIS
LIN {X 58.3027,Y 46.8749,Z 77,A 33.5444,B 24.8863,C -2.4613,E1 25.1236,E2 410.8205} C_DIS
LIN {X 56.3332,Y 49.2235,Z 77,A 36.033,B 24.8854,C -2.4708,E1 25.1191,E2 408.3207} C_DIS
LIN {X 53.9987,Y 51.7742,Z 77,A 38.5706,B 24.8852,C -2.4733,E1 25.1142,E2 405.7882} C_DIS
LIN {X 51.6823,Y 54.087,Z 77,A 41.3854,B 24.8839,C -2.4874,E1 25.1085,E2 402.9518} C_DIS
LIN {X 49.0139,Y 56.5163,Z 77,A 43.799,B 24.8843,C -2.4827,E1 25.1035,E2 400.559} C_DIS
LIN {X 46.6597,Y 58.4754,Z 77,A 46.0804,B 24.8841,C -2.4852,E1 25.0986,E2 398.2803} C_DIS
LIN {X 43.9154,Y 60.5635,Z 77,A 48.7911,B 24.8835,C -2.4918,E1 25.0925,E2 395.5638} C_DIS
LIN {X 41.2742,Y 62.3926,Z 77,A 51.1359,B 24.8834,C -2.4925,E1 25.0871,E2 393.2252} C_DIS
LIN {X 37.6404,Y 64.6507,Z 77,A 54.5883,B 24.8825,C -2.5022,E1 25.0788,E2 389.7605} C_DIS
LIN {X 34.7643,Y 66.2408,Z 77,A 56.8788,B 24.8828,C -2.4992,E1 25.0732,E2 387.4836} C_DIS
LIN {X 32.3188,Y 67.4677,Z 77,A 59.0104,B 24.8824,C -2.5028,E1 25.0679,E2 385.3492} C_DIS
LIN {X 29.4086,Y 68.7871,Z 77,A 61.2264,B 24.8828,C -2.4991,E1 25.0623,E2 383.1475} C_DIS
LIN {X 27.257,Y 69.6667,Z 77,A 63.2489,B 24.882,C -2.5076,E1 25.057,E2 381.1094} C_DIS
LIN {X 24.2818,Y 70.7597,Z 77,A 65.7367,B 24.8816,C -2.5113,E1 25.0504,E2 378.6177} C_DIS
LIN {X 20.2889,Y 72.0052,Z 77,A 68.8067,B 24.8817,C -2.51,E1 25.0422,E2 375.5563} C_DIS
LIN {X 17.4855,Y 72.7372,Z 77,A 71.4379,B 24.8806,C -2.5225,E1 25.035,E2 372.8992} C_DIS
LIN {X 13.4869,Y 73.5836,Z 77,A 74.272,B 24.8812,C -2.5158,E1 25.0273,E2 370.0846} C_DIS
LIN {X 10.0802,Y 74.128,Z 77,A 76.8036,B 24.8814,C -2.5135,E1 25.0204,E2 367.5607} C_DIS
LIN {X 7.7378,Y 74.4077,Z 77,A 78.8371,B 24.8808,C -2.5199,E1 25.0147,E2 365.5135} C_DIS
LIN {X 3.6605,Y 74.7207,Z 77,A 81.8965,B 24.881,C -2.5179,E1 25.0062,E2 362.46} C_DIS
LIN {X 0.3491,Y 74.8082,Z 77,A 84.3334,B 24.8813,C -2.5149,E1 24.9994,E2 360.0305} C_DIS
LIN {X -2.6088,Y 74.7641,Z 77,A 87.0033,B 24.8803,C -2.525,E1 24.9919,E2 357.3365} C_DIS
LIN {X -5.7998,Y 74.584,Z 77,A 89.0161,B 24.8815,C -2.5125,E1 24.9863,E2 355.3525} C_DIS
LIN {X -9.8036,Y 74.1641,Z 77,A 91.8747,B 24.8822,C -2.505,E1 24.9785,E2 352.5099} C_DIS
LIN {X -11.6215,Y 73.901,Z 77,A 93.619,B 24.8815,C -2.5128,E1 24.9736,E2 350.7457} C_DIS
LIN {X -14.8129,Y 73.3281,Z 77,A 96.0509,B 24.8818,C -2.5095,E1 24.9669,E2 348.3189} C_DIS
LIN {X -17.5118,Y 72.7308,Z 77,A 98.4404,B 24.8813,C -2.5145,E1 24.9604,E2 345.9142} C_DIS
LIN {X -21.1136,Y 71.7679,Z 77,A 101.0404,B 24.8822,C -2.505,E1 24.9534,E2 343.3327} C_DIS
LIN {X -25.0017,Y 70.5078,Z 77,A 104.1609,B 24.8826,C -2.501,E1 24.9452,E2 340.2159} C_DIS
LIN {X -27.7209,Y 69.4845,Z 77,A 106.5233,B 24.8826,C -2.5015,E1 24.939,E2 337.8473} C_DIS
LIN {X -31.0389,Y 68.0667,Z 77,A 109.2026,B 24.8831,C -2.4954,E1 24.9322,E2 335.1762} C_DIS
LIN {X -33.5545,Y 66.8626,Z 77,A 111.2855,B 24.8836,C -2.4907,E1 24.927,E2 333.099} C_DIS
LIN {X -36.0731,Y 65.5387,Z 77,A 113.3091,B 24.8843,C -2.4832,E1 24.9221,E2 331.0876} C_DIS
LIN {X -38.0499,Y 64.4095,Z 77,A 115.2616,B 24.8841,C -2.4853,E1 24.9173,E2 329.1243} C_DIS
LIN {X -40.7833,Y 62.716,Z 77,A 117.7658,B 24.8844,C -2.4817,E1 24.9114,E2 326.6206} C_DIS
LIN {X -43.2878,Y 61.013,Z 77,A 120.1016,B 24.8848,C -2.4775,E1 24.9061,E2 324.2867} C_DIS
LIN {X -45.9271,Y 59.0525,Z 77,A 122.4801,B 24.8856,C -2.4689,E1 24.9008,E2 321.9203} C_DIS
LIN {X -49.493,Y 56.0978,Z 77,A 126.7989,B 24.8846,C -2.4799,E1 24.8915,E2 317.5584} C_DIS
LIN {X -51.8704,Y 53.9059,Z 77,A 128.6746,B 24.8865,C -2.4595,E1 24.8878,E2 315.7237} C_DIS
LIN {X -54.16,Y 51.6067,Z 77,A 131.1787,B 24.887,C -2.454,E1 24.883,E2 313.2221} C_DIS
LIN {X -56.176,Y 49.4034,Z 77,A 133.4999,B 24.8874,C -2.4491,E1 24.8786,E2 310.9021} C_DIS
LIN {X -58.3053,Y 46.8718,Z 77,A 136.0182,B 24.8881,C -2.4422,E1 24.8742,E2 308.3886} C_DIS
LIN {X -60.164,Y 44.461,Z 77,A 138.1466,B 24.8891,C -2.4312,E1 24.8706,E2 306.2764} C_DIS
LIN {X -61.2286,Y 42.9832,Z 77,A 139.7671,B 24.8889,C -2.4328,E1 24.868,E2 304.6441} C_DIS
LIN {X -62.8896,Y 40.513,Z 77,A 142.0515,B 24.8895,C -2.4266,E1 24.8645,E2 302.363} C_DIS
LIN {X -64.5264,Y 37.8522,Z 77,A 144.5622,B 24.8899,C -2.4226,E1 24.8609,E2 299.8488} C_DIS
LIN {X -66.7767,Y 33.725,Z 77,A 147.8318,B 24.8915,C -2.4044,E1 24.8566,E2 296.6055} C_DIS
LIN {X -67.7554,Y 31.7114,Z 77,A 149.7466,B 24.8915,C -2.404,E1 24.8543,E2 294.681} C_DIS
LIN {X -68.922,Y 29.0885,Z 77,A 152.0627,B 24.8919,C -2.4002,E1 24.8517,E2 292.3612} C_DIS
LIN {X -70.3719,Y 25.3822,Z 77,A 155.1097,B 24.8927,C -2.3909,E1 24.8487,E2 289.3193} C_DIS
LIN {X -71.3686,Y 22.4274,Z 77,A 157.4686,B 24.8934,C -2.3829,E1 24.8467,E2 286.9661} C_DIS
LIN {X -72.1222,Y 19.8694,Z 77,A 159.6177,B 24.8938,C -2.3791,E1 24.8451,E2 284.8137} C_DIS
LIN {X -72.9178,Y 16.715,Z 77,A 162.1329,B 24.8944,C -2.3718,E1 24.8434,E2 282.3011} C_DIS
LIN {X -73.6679,Y 13.0184,Z 77,A 164.7435,B 24.8958,C -2.3562,E1 24.8421,E2 279.7125} C_DIS
LIN {X -74.2239,Y 9.3418,Z 77,A 168.3603,B 24.895,C -2.3652,E1 24.8407,E2 276.0525} C_DIS
LIN {X -74.7178,Y 3.7089,Z 77,A 172.4872,B 24.8967,C -2.3466,E1 24.8399,E2 271.9452} C_DIS
LIN {X -74.8083,Y 0.277,Z 77,A 174.608,B 24.8985,C -2.3263,E1 24.8398,E2 269.86} C_DIS
LIN {X -74.7621,Y -2.6454,Z 77,A 177.1577,B 24.8985,C -2.3265,E1 24.84,E2 267.2945} C_DIS
LIN {X -74.548,Y -6.2466,Z 77,A -179.8261,B 24.8987,C -2.3238,E1 24.8406,E2 264.2667} C_DIS
LIN {X -74.2043,Y -9.4929,Z 77,A -176.9886,B 24.8987,C -2.324,E1 24.8416,E2 261.4118} C_DIS
LIN {X -73.7243,Y -12.6984,Z 77,A -174.4565,B 24.8992,C -2.3175,E1 24.8428,E2 258.8801} C_DIS
LIN {X -73.1016,Y -15.8914,Z 77,A -172.8035,B 24.9016,C -2.29,E1 24.8437,E2 257.2831} C_DIS
LIN {X -72.5858,Y -18.106,Z 77,A -170.8881,B 24.9017,C -2.2888,E1 24.8449,E2 255.3593} C_DIS
LIN {X -72.0674,Y -20.0694,Z 77,A -169.2707,B 24.902,C -2.2856,E1 24.8461,E2 253.7402} C_DIS
LIN {X -71.2234,Y -22.8829,Z 77,A -167.0607,B 24.9026,C -2.278,E1 24.848,E2 251.5357} C_DIS
LIN {X -70.3169,Y -25.5329,Z 77,A -164.9584,B 24.9033,C -2.2707,E1 24.8499,E2 249.4388} C_DIS
LIN {X -68.76,Y -29.4729,Z 77,A -161.5446,B 24.9037,C -2.2654,E1 24.8535,E2 246.0186} C_DIS
LIN {X -67.5401,Y -32.1679,Z 77,A -159.2703,B 24.9042,C -2.2594,E1 24.8562,E2 243.7464} C_DIS
LIN {X -65.6172,Y -35.9284,Z 77,A -156.0647,B 24.905,C -2.2499,E1 24.8603,E2 240.5463} C_DIS
LIN {X -64.1671,Y -38.46,Z 77,A -153.7832,B 24.9054,C -2.2451,E1 24.8636,E2 238.2644} C_DIS
LIN {X -62.685,Y -40.8295,Z 77,A -151.2687,B 24.9051,C -2.2488,E1 24.8674,E2 235.7284} C_DIS
LIN {X -59.6879,Y -45.0974,Z 77,A -147.8438,B 24.9071,C -2.2251,E1 24.8729,E2 232.3433} C_DIS
LIN {X -58.5628,Y -46.5492,Z 77,A -146.4295,B 24.9074,C -2.222,E1 24.8754,E2 230.9298} C_DIS
LIN {X -57.3493,Y -48.0367,Z 77,A -144.7039,B 24.9071,C -2.2248,E1 24.8785,E2 229.1894} C_DIS
LIN {X -55.2481,Y -50.4388,Z 77,A -142.3267,B 24.9077,C -2.2178,E1 24.8829,E2 226.8185} C_DIS
LIN {X -53.4584,Y -52.3321,Z 77,A -139.7678,B 24.9069,C -2.2275,E1 24.8879,E2 224.2253} C_DIS
LIN {X -48.843,Y -56.665,Z 77,A -135.0818,B 24.9081,C -2.2139,E1 24.8976,E2 219.5531} C_DIS
LIN {X -46.7186,Y -58.4289,Z 77,A -133.225,B 24.9089,C -2.2035,E1 24.9016,E2 217.714} C_DIS
LIN {X -44.1997,Y -60.3553,Z 77,A -130.845,B 24.9094,C -2.1982,E1 24.9069,E2 215.3383} C_DIS
LIN {X -41.6458,Y -62.1461,Z 77,A -128.4567,B 24.9097,C -2.1943,E1 24.9124,E2 212.9512} C_DIS
LIN {X -38.9025,Y -63.8982,Z 77,A -126.0449,B 24.9102,C -2.1885,E1 24.9181,E2 210.5455} C_DIS
LIN {X -36.4216,Y -65.3441,Z 77,A -123.6788,B 24.9101,C -2.1897,E1 24.9239,E2 208.1695} C_DIS
LIN {X -33.7177,Y -66.7805,Z 77,A -121.2663,B 24.9101,C -2.1885,E1 24.9299,E2 205.7534} C_DIS
LIN {X -30.6897,Y -68.2241,Z 77,A -118.8461,B 24.9107,C -2.1818,E1 24.936,E2 203.3431} C_DIS
LIN {X -27.6888,Y -69.4971,Z 77,A -116.3197,B 24.9109,C -2.1801,E1 24.9425,E2 200.8152} C_DIS
LIN {X -23.8926,Y -70.8909,Z 77,A -113.5931,B 24.9119,C -2.1677,E1 24.9496,E2 198.1124} C_DIS
LIN {X -21.8601,Y -71.5445,Z 77,A -111.5845,B 24.9112,C -2.1763,E1 24.955,E2 196.0799} C_DIS
LIN {X -18.6735,Y -72.4409,Z 77,A -109.1994,B 24.9116,C -2.1708,E1 24.9614,E2 193.7042} C_DIS
LIN {X -16.6711,Y -72.928,Z 77,A -107.4014,B 24.9112,C -2.1758,E1 24.9664,E2 191.8919} C_DIS
LIN {X -13.7655,Y -73.5326,Z 77,A -105.2079,B 24.9114,C -2.1728,E1 24.9723,E2 189.7032} C_DIS
LIN {X -11.0285,Y -73.9927,Z 77,A -102.8654,B 24.911,C -2.178,E1 24.9789,E2 187.3461} C_DIS
LIN {X -7.347,Y -74.4486,Z 77,A -100.0956,B 24.9112,C -2.1758,E1 24.9865,E2 184.58} C_DIS
LIN {X -3.7377,Y -74.7166,Z 77,A -97.4482,B 24.9115,C -2.1725,E1 24.9939,E2 181.9395} C_DIS
LIN {X -1.1871,Y -74.7998,Z 77,A -95.6051,B 24.9117,C -2.1698,E1 24.999,E2 180.1026} C_DIS
LIN {X 0.4964,Y -74.8047,Z 77,A -94.4275,B 24.9119,C -2.1671,E1 25.0023,E2 178.9315} C_DIS
Enddeposition()
LIN {X 0.4964,Y -74.8047,Z 77,A -94.4275,B 24.9119,C -2.1671,E1 25.0023,E2 178.9315} C_DIS
Startdeposition()
$VEL.CP = VEL_PRINT
LIN {X -0.6606,Y -73.8541,Z 77,A -96.2607,B 24.9126,C -2.1584,E1 24.9971,E2 180.7852} C_DIS
LIN {X -3.8104,Y -73.7589,Z 77,A -98.5659,B 24.9123,C -2.1618,E1 24.9907,E2 183.0828} C_DIS
LIN {X -5.9258,Y -73.6186,Z 77,A -100.4807,B 24.9129,C -2.1548,E1 24.9853,E2 185.015} C_DIS
LIN {X -10.7353,Y -73.0732,Z 77,A -104.0808,B 24.9125,C -2.1594,E1 24.9754,E2 188.6067} C_DIS
LIN {X -13.7658,Y -72.5628,Z 77,A -106.3677,B 24.9123,C -2.1627,E1 24.9691,E2 190.8881} C_DIS
LIN {X -15.6488,Y -72.1799,Z 77,A -107.9568,B 24.9124,C -2.1609,E1 24.9647,E2 192.4836} C_DIS
LIN {X -20.8311,Y -70.8584,Z 77,A -112.6047,B 24.9132,C -2.1508,E1 24.9521,E2 197.1626} C_DIS
LIN {X -26.1751,Y -69.0629,Z 77,A -116.3219,B 24.9116,C -2.1709,E1 24.9424,E2 200.8391} C_DIS
LIN {X -28.6017,Y -68.0938,Z 77,A -118.3889,B 24.9116,C -2.1719,E1 24.9371,E2 202.9083} C_DIS
LIN {X -30.8624,Y -67.1003,Z 77,A -120.3562,B 24.9115,C -2.1727,E1 24.9321,E2 204.8785} C_DIS
LIN {X -34.4384,Y -65.3362,Z 77,A -123.5299,B 24.9113,C -2.1745,E1 24.9242,E2 208.0564} C_DIS
LIN {X -37.1287,Y -63.8469,Z 77,A -126.7132,B 24.9126,C -2.1583,E1 24.9163,E2 211.2877} C_DIS
LIN {X -40.259,Y -61.921,Z 77,A -128.899,B 24.911,C -2.1788,E1 24.9113,E2 213.4317} C_DIS
LIN {X -43.2673,Y -59.8573,Z 77,A -131.741,B 24.9106,C -2.1832,E1 24.9048,E2 216.2731} C_DIS
LIN {X -45.9514,Y -57.8215,Z 77,A -134.1842,B 24.9099,C -2.1919,E1 24.8994,E2 218.7044} C_DIS
LIN {X -48.1779,Y -55.9808,Z 77,A -136.5694,B 24.9099,C -2.1926,E1 24.8943,E2 221.097} C_DIS
LIN {X -50.7519,Y -53.6573,Z 77,A -139.3025,B 24.9095,C -2.197,E1 24.8887,E2 223.8309} C_DIS
LIN {X -53.5798,Y -50.8344,Z 77,A -142.3977,B 24.9089,C -2.2036,E1 24.8827,E2 226.9236} C_DIS
LIN {X -55.9521,Y -48.2116,Z 77,A -145.1572,B 24.9084,C -2.2094,E1 24.8776,E2 229.6817} C_DIS
LIN {X -58.3474,Y -45.282,Z 77,A -148.4194,B 24.9084,C -2.2086,E1 24.8719,E2 232.9611} C_DIS
LIN {X -61.2795,Y -41.2273,Z 77,A -152.3598,B 24.9078,C -2.2169,E1 24.8656,E2 236.9012} C_DIS
LIN {X -63.5827,Y -37.5774,Z 77,A -155.3451,B 24.9064,C -2.234,E1 24.8613,E2 239.861} C_DIS
LIN {X -66.22,Y -32.7069,Z 77,A -159.4678,B 24.9051,C -2.2496,E1 24.8559,E2 243.9682} C_DIS
LIN {X -67.8056,Y -29.2794,Z 77,A -162.8892,B 24.9053,C -2.2465,E1 24.852,E2 247.4157} C_DIS
LIN {X -69.1014,Y -26.0734,Z 77,A -165.1813,B 24.9039,C -2.2632,E1 24.8497,E2 249.681} C_DIS
LIN {X -70.078,Y -23.3232,Z 77,A -167.5726,B 24.9036,C -2.2669,E1 24.8475,E2 252.077} C_DIS
LIN {X -71.0097,Y -20.3096,Z 77,A -170.3497,B 24.9036,C -2.2667,E1 24.8453,E2 254.8707} C_DIS
LIN {X -72.0828,Y -16.0942,Z 77,A -173.126,B 24.9016,C -2.2905,E1 24.8435,E2 257.6063} C_DIS
LIN {X -73.0832,Y -10.6616,Z 77,A -177.8436,B 24.9013,C -2.2939,E1 24.8412,E2 262.3438} C_DIS
LIN {X -73.4543,Y -7.6995,Z 77,A 179.3637,B 24.9016,C -2.2904,E1 24.8404,E2 265.1615} C_DIS
LIN {X -73.7862,Y -3.2286,Z 77,A 176.5121,B 24.8994,C -2.3155,E1 24.8399,E2 267.9704} C_DIS
LIN {X -73.8571,Y 0.0518,Z 77,A 173.5585,B 24.8995,C -2.3144,E1 24.8399,E2 270.9445} C_DIS
LIN {X -73.6574,Y 5.4328,Z 77,A 169.6973,B 24.8977,C -2.3347,E1 24.8403,E2 274.7802} C_DIS
LIN {X -73.2919,Y 9.124,Z 77,A 166.4381,B 24.8977,C -2.3353,E1 24.8414,E2 278.0576} C_DIS
LIN {X -72.7445,Y 12.773,Z 77,A 163.9001,B 24.8962,C -2.3516,E1 24.8425,E2 280.5717} C_DIS
LIN {X -71.9857,Y 16.5194,Z 77,A 160.7013,B 24.8959,C -2.3557,E1 24.8444,E2 283.7796} C_DIS
LIN {X -70.8552,Y 20.8419,Z 77,A 157.5218,B 24.8943,C -2.373,E1 24.8467,E2 286.9363} C_DIS
LIN {X -70.1177,Y 23.2052,Z 77,A 155.7335,B 24.8935,C -2.3819,E1 24.8482,E2 288.7136} C_DIS
LIN {X -69.4481,Y 25.1359,Z 77,A 153.0397,B 24.8953,C -2.3618,E1 24.8508,E2 291.4707} C_DIS
LIN {X -68.0732,Y 28.6507,Z 77,A 151.2864,B 24.8922,C -2.3971,E1 24.8526,E2 293.1494} C_DIS
LIN {X -65.9934,Y 33.164,Z 77,A 147.2007,B 24.8916,C -2.4032,E1 24.8575,E2 297.2428} C_DIS
LIN {X -64.9894,Y 35.0886,Z 77,A 145.0277,B 24.8922,C -2.3969,E1 24.8603,E2 299.4422} C_DIS
LIN {X -62.9927,Y 38.5589,Z 77,A 142.3395,B 24.8905,C -2.4152,E1 24.8641,E2 302.1007} C_DIS
LIN {X -61.3529,Y 41.1188,Z 77,A 139.9195,B 24.8901,C -2.4203,E1 24.8678,E2 304.5206} C_DIS
LIN {X -59.541,Y 43.7001,Z 77,A 137.3702,B 24.8897,C -2.4246,E1 24.8719,E2 307.0722} C_DIS
LIN {X -57.8827,Y 45.874,Z 77,A 135.3481,B 24.889,C -2.4324,E1 24.8754,E2 309.0852} C_DIS
LIN {X -56.1649,Y 47.9618,Z 77,A 133.1939,B 24.8886,C -2.4365,E1 24.8793,E2 311.2396} C_DIS
LIN {X -54.0898,Y 50.292,Z 77,A 130.6655,B 24.8883,C -2.44,E1 24.884,E2 313.7709} C_DIS
LIN {X -51.9032,Y 52.5441,Z 77,A 128.3601,B 24.8875,C -2.4488,E1 24.8885,E2 316.065} C_DIS
LIN {X -48.8858,Y 55.3639,Z 77,A 124.5077,B 24.8882,C -2.441,E1 24.8966,E2 319.9515} C_DIS
LIN {X -45.2425,Y 58.3778,Z 77,A 121.2085,B 24.8867,C -2.4575,E1 24.9037,E2 323.2238} C_DIS
LIN {X -42.3436,Y 60.5136,Z 77,A 118.6111,B 24.8857,C -2.4677,E1 24.9095,E2 325.8058} C_DIS
LIN {X -40.2514,Y 61.9259,Z 77,A 116.5286,B 24.8857,C -2.4685,E1 24.9144,E2 327.8933} C_DIS
LIN {X -37.5647,Y 63.5902,Z 77,A 114.475,B 24.8843,C -2.4825,E1 24.9192,E2 329.9199} C_DIS
LIN {X -35.6147,Y 64.7041,Z 77,A 111.7654,B 24.8862,C -2.4623,E1 24.926,E2 332.6853} C_DIS
LIN {X -31.5608,Y 66.7752,Z 77,A 108.7395,B 24.8846,C -2.48,E1 24.9335,E2 335.6771} C_DIS
LIN {X -28.3328,Y 68.2071,Z 77,A 106.2437,B 24.8836,C -2.4898,E1 24.9398,E2 338.1553} C_DIS
LIN {X -26.5045,Y 68.9382,Z 77,A 103.5195,B 24.8861,C -2.4629,E1 24.9471,E2 340.9493} C_DIS
LIN {X -22.4408,Y 70.3657,Z 77,A 101.226,B 24.8834,C -2.4923,E1 24.953,E2 343.1772} C_DIS
LIN {X -20.4537,Y 70.9688,Z 77,A 99.6171,B 24.8832,C -2.494,E1 24.9573,E2 344.7845} C_DIS
LIN {X -14.5262,Y 72.4149,Z 77,A 94.7868,B 24.8831,C -2.4959,E1 24.9705,E2 349.6167} C_DIS
LIN {X -7.4537,Y 73.4801,Z 77,A 89.548,B 24.882,C -2.5073,E1 24.9849,E2 354.8327} C_DIS
LIN {X -4.1307,Y 73.7412,Z 77,A 86.2209,B 24.8837,C -2.4896,E1 24.9943,E2 358.2029} C_DIS
LIN {X -0.9599,Y 73.8516,Z 77,A 83.27,B 24.8848,C -2.4778,E1 25.0026,E2 361.182} C_DIS
LIN {X 3.1336,Y 73.7902,Z 77,A 81.2168,B 24.8821,C -2.5067,E1 25.0082,E2 363.1662} C_DIS
LIN {X 7.9386,Y 73.4293,Z 77,A 77.301,B 24.8825,C -2.5018,E1 25.0191,E2 367.0914} C_DIS
LIN {X 10.6172,Y 73.09,Z 77,A 75.0492,B 24.8829,C -2.4972,E1 25.0253,E2 369.3522} C_DIS
LIN {X 13.6301,Y 72.5889,Z 77,A 72.1048,B 24.8844,C -2.4814,E1 25.0335,E2 372.3308} C_DIS
LIN {X 17.108,Y 71.8487,Z 77,A 70.3819,B 24.882,C -2.5071,E1 25.038,E2 373.9905} C_DIS
LIN {X 20.2078,Y 71.0385,Z 77,A 67.2234,B 24.8838,C -2.4877,E1 25.0466,E2 377.1898} C_DIS
LIN {X 23.9172,Y 69.8777,Z 77,A 64.6239,B 24.883,C -2.4963,E1 25.0535,E2 379.7641} C_DIS
LIN {X 26.3796,Y 68.9854,Z 77,A 62.6063,B 24.8832,C -2.4948,E1 25.0587,E2 381.7809} C_DIS
LIN {X 28.8643,Y 67.9832,Z 77,A 60.2295,B 24.8841,C -2.4846,E1 25.0649,E2 384.1762} C_DIS
LIN {X 32.1443,Y 66.4951,Z 77,A 57.6617,B 24.8839,C -2.4875,E1 25.0714,E2 386.7307} C_DIS
LIN {X 34.8535,Y 65.117,Z 77,A 54.8242,B 24.8854,C -2.4714,E1 25.0784,E2 389.5983} C_DIS
LIN {X 39.4041,Y 62.4679,Z 77,A 51.3731,B 24.8843,C -2.4827,E1 25.0866,E2 393.012} C_DIS
LIN {X 41.5725,Y 61.0458,Z 77,A 49.3512,B 24.8846,C -2.4792,E1 25.0913,E2 395.0354} C_DIS
LIN {X 43.4221,Y 59.7445,Z 77,A 46.8724,B 24.8868,C -2.4563,E1 25.097,E2 397.5595} C_DIS
LIN {X 46.1033,Y 57.7015,Z 77,A 44.4142,B 24.8868,C -2.4559,E1 25.1024,E2 400.0097} C_DIS
LIN {X 50.4435,Y 53.9471,Z 77,A 40.5233,B 24.8862,C -2.4627,E1 25.1104,E2 403.8689} C_DIS
LIN {X 52.518,Y 51.9296,Z 77,A 38.336,B 24.8865,C -2.4596,E1 25.1147,E2 406.0542} C_DIS
LIN {X 54.5291,Y 49.8139,Z 77,A 35.3978,B 24.8886,C -2.4358,E1 25.1204,E2 409.0358} C_DIS
LIN {X 56.6457,Y 47.3935,Z 77,A 33.9017,B 24.8866,C -2.4582,E1 25.123,E2 410.4722} C_DIS
LIN {X 58.6949,Y 44.8311,Z 77,A 30.5975,B 24.8891,C -2.4307,E1 25.1288,E2 413.826} C_DIS
LIN {X 61.1666,Y 41.394,Z 77,A 27.8519,B 24.8885,C -2.4378,E1 25.1331,E2 416.5412} C_DIS
LIN {X 62.7532,Y 38.9473,Z 77,A 25.1096,B 24.8902,C -2.4183,E1 25.1373,E2 419.3158} C_DIS
LIN {X 65.1264,Y 34.8362,Z 77,A 21.7313,B 24.8904,C -2.4171,E1 25.1418,E2 422.6792} C_DIS
LIN {X 66.8129,Y 31.4798,Z 77,A 18.6179,B 24.8916,C -2.4034,E1 25.1456,E2 425.8085} C_DIS
LIN {X 68.4755,Y 27.6759,Z 77,A 15.7141,B 24.8916,C -2.4034,E1 25.1488,E2 428.6965} C_DIS
LIN {X 69.5438,Y 24.8731,Z 77,A 12.3078,B 24.895,C -2.3656,E1 25.1521,E2 432.1728} C_DIS
LIN {X 70.9439,Y 20.5416,Z 77,A 9.8194,B 24.8933,C -2.385,E1 25.154,E2 434.6012} C_DIS
LIN {X 71.6269,Y 18.0153,Z 77,A 7.638,B 24.8942,C -2.3745,E1 25.1555,E2 436.7949} C_DIS
LIN {X 72.5068,Y 14.0567,Z 77,A 4.2623,B 24.8957,C -2.3582,E1 25.1574,E2 440.1894} C_DIS
LIN {X 73.2339,Y 9.5715,Z 77,A 1.2639,B 24.8953,C -2.3625,E1 25.1586,E2 443.1599} C_DIS
LIN {X 73.5181,Y 7.0706,Z 77,A -1.036,B 24.8967,C -2.3463,E1 25.1593,E2 445.4845} C_DIS
LIN {X 73.8403,Y 1.5756,Z 77,A -4.9596,B 24.897,C -2.3429,E1 25.1598,E2 449.3929} C_DIS
LIN {X 73.8424,Y -1.4586,Z 77,A -8.0434,B 24.8995,C -2.3142,E1 25.1596,E2 452.5261} C_DIS
LIN {X 73.6776,Y -5.1433,Z 77,A -9.9278,B 24.8978,C -2.3335,E1 25.1593,E2 454.3537} C_DIS
LIN {X 73.2341,Y -9.5702,Z 77,A -13.5902,B 24.8993,C -2.3163,E1 25.1582,E2 458.035} C_DIS
LIN {X 72.775,Y -12.6014,Z 77,A -15.8967,B 24.8998,C -2.3109,E1 25.1572,E2 460.3408} C_DIS
LIN {X 72.2422,Y -15.3631,Z 77,A -18.0974,B 24.9005,C -2.3034,E1 25.1559,E2 462.5462} C_DIS
LIN {X 70.9523,Y -20.5121,Z 77,A -22.5312,B 24.9024,C -2.2813,E1 25.1527,E2 467.0066} C_DIS
LIN {X 69.6198,Y -24.6566,Z 77,A -25.5026,B 24.9022,C -2.2828,E1 25.1501,E2 469.9579} C_DIS
LIN {X 67.9849,Y -28.8601,Z 77,A -29.0169,B 24.9032,C -2.2717,E1 25.1465,E2 473.4789} C_DIS
LIN {X 66.6622,Y -31.7964,Z 77,A -31.3912,B 24.9035,C -2.2679,E1 25.1437,E2 475.8494} C_DIS
LIN {X 65.5834,Y -33.9677,Z 77,A -33.5187,B 24.9046,C -2.2552,E1 25.141,E2 477.9956} C_DIS
LIN {X 63.962,Y -36.9283,Z 77,A -36.2032,B 24.9054,C -2.2458,E1 25.1373,E2 480.6884} C_DIS
LIN {X 61.8523,Y -40.3637,Z 77,A -39.3072,B 24.9061,C -2.2377,E1 25.1326,E2 483.7959} C_DIS
LIN {X 58.8665,Y -44.6054,Z 77,A -43.5648,B 24.9075,C -2.2201,E1 25.1256,E2 488.0743} C_DIS
LIN {X 55.405,Y -48.8387,Z 77,A -47.3203,B 24.9073,C -2.2232,E1 25.1188,E2 491.8056} C_DIS
LIN {X 52.6993,Y -51.7461,Z 77,A -50.3361,B 24.9078,C -2.2175,E1 25.113,E2 494.8217} C_DIS
LIN {X 50.6839,Y -53.7213,Z 77,A -52.694,B 24.9086,C -2.2075,E1 25.1082,E2 497.1935} C_DIS
LIN {X 48.0865,Y -56.0586,Z 77,A -55.4255,B 24.9091,C -2.2008,E1 25.1025,E2 499.9301} C_DIS
LIN {X 44.1666,Y -59.1962,Z 77,A -58.7583,B 24.9085,C -2.2084,E1 25.0953,E2 503.2326} C_DIS
LIN {X 40.348,Y -61.8625,Z 77,A -62.3805,B 24.9091,C -2.2009,E1 25.0869,E2 506.8602} C_DIS
LIN {X 36.3097,Y -64.316,Z 77,A -66.2606,B 24.9102,C -2.1881,E1 25.0776,E2 510.7583} C_DIS
LIN {X 33.1495,Y -66.0006,Z 77,A -68.8197,B 24.9101,C -2.1896,E1 25.0713,E2 513.3069} C_DIS
LIN {X 30.6225,Y -67.2099,Z 77,A -71.6122,B 24.9118,C -2.1691,E1 25.0641,E2 516.1408} C_DIS
LIN {X 26.7602,Y -68.8388,Z 77,A -74.5634,B 24.9115,C -2.1727,E1 25.0565,E2 519.0766} C_DIS
LIN {X 23.9517,Y -69.8661,Z 77,A -76.5855,B 24.911,C -2.178,E1 25.0512,E2 521.0823} C_DIS
LIN {X 21.9866,Y -70.5082,Z 77,A -78.6793,B 24.9123,C -2.1627,E1 25.0456,E2 523.2084} C_DIS
LIN {X 18.8382,Y -71.4144,Z 77,A -81.2302,B 24.9125,C -2.1597,E1 25.0387,E2 525.7621} C_DIS
LIN {X 15.5236,Y -72.2072,Z 77,A -83.3394,B 24.9115,C -2.1718,E1 25.033,E2 527.84} C_DIS
LIN {X 11.312,Y -72.9853,Z 77,A -86.8203,B 24.9121,C -2.1649,E1 25.0234,E2 531.3334} C_DIS
LIN {X 8.4804,Y -73.3683,Z 77,A -89.0185,B 24.9121,C -2.164,E1 25.0173,E2 533.532} C_DIS
LIN {X 4.1089,Y -73.7424,Z 77,A -92.4086,B 24.9123,C -2.1627,E1 25.0079,E2 536.9234} C_DIS
LIN {X 0.4828,Y -73.8381,Z 77,A -94.3735,B 24.9105,C -2.1847,E1 25.0026,E2 538.8355} C_DIS
Enddeposition()
LIN {X 0.4828,Y -73.8381,Z 77,A -94.3735,B 24.9105,C -2.1847,E1 25.0026,E2 538.8355} C_DIS
Startdeposition()
$VEL.CP = VEL_PRINT
LIN {X 1.2599,Y -72.8937,Z 77,A -93.2818,B 24.9081,C -2.2138,E1 25.0058,E2 537.6751} C_DIS
LIN {X 4.1876,Y -72.7843,Z 77,A -90.9676,B 24.908,C -2.215,E1 25.0123,E2 535.3588} C_DIS
LIN {X 9.1535,Y -72.3279,Z 77,A -87.4324,B 24.9086,C -2.2069,E1 25.022,E2 531.8454} C_DIS
LIN {X 13.6721,Y -71.6111,Z 77,A -83.8294,B 24.9084,C -2.2098,E1 25.0319,E2 528.2391} C_DIS
LIN {X 17.86,Y -70.6836,Z 77,A -80.4132,B 24.908,C -2.2142,E1 25.0412,E2 524.8173} C_DIS
LIN {X 19.9023,Y -70.1354,Z 77,A -77.9807,B 24.9061,C -2.2373,E1 25.0479,E2 522.3341} C_DIS
LIN {X 23.5027,Y -69.0126,Z 77,A -75.8048,B 24.9076,C -2.2191,E1 25.0535,E2 520.2057} C_DIS
LIN {X 26.5981,Y -67.8794,Z 77,A -73.387,B 24.9077,C -2.2177,E1 25.0598,E2 517.7961} C_DIS
LIN {X 29.7339,Y -66.5659,Z 77,A -70.5254,B 24.907,C -2.2269,E1 25.0672,E2 514.9196} C_DIS
LIN {X 32.0938,Y -65.4611,Z 77,A -68.1371,B 24.9059,C -2.2397,E1 25.0733,E2 512.5073} C_DIS
LIN {X 36.1212,Y -63.3276,Z 77,A -64.2197,B 24.9046,C -2.2555,E1 25.0829,E2 508.5641} C_DIS
LIN {X 39.2188,Y -61.4572,Z 77,A -62.3053,B 24.9063,C -2.2345,E1 25.0873,E2 506.7057} C_DIS
LIN {X 42.993,Y -58.8785,Z 77,A -58.6977,B 24.9057,C -2.2421,E1 25.0956,E2 503.0925} C_DIS
LIN {X 46.2325,Y -56.3685,Z 77,A -55.3278,B 24.9048,C -2.2533,E1 25.103,E2 499.7087} C_DIS
LIN {X 49.2826,Y -53.7237,Z 77,A -51.7363,B 24.9031,C -2.2725,E1 25.1105,E2 496.0859} C_DIS
LIN {X 53.1484,Y -49.9031,Z 77,A -47.651,B 24.9027,C -2.2775,E1 25.1185,E2 492.0064} C_DIS
LIN {X 54.9724,Y -47.8865,Z 77,A -44.7438,B 24.9003,C -2.3054,E1 25.1239,E2 489.0462} C_DIS
LIN {X 57.8373,Y -44.3839,Z 77,A -42.3727,B 24.9025,C -2.2802,E1 25.1278,E2 486.7461} C_DIS
LIN {X 60.0707,Y -41.3104,Z 77,A -39.1874,B 24.9013,C -2.2941,E1 25.133,E2 483.5434} C_DIS
LIN {X 62.0096,Y -38.3395,Z 77,A -36.467,B 24.9008,C -2.2999,E1 25.1371,E2 480.8229} C_DIS
LIN {X 63.9589,Y -34.9915,Z 77,A -33.1432,B 24.8993,C -2.3169,E1 25.1416,E2 477.4764} C_DIS
LIN {X 65.7206,Y -31.5574,Z 77,A -30.4799,B 24.8995,C -2.3149,E1 25.1449,E2 474.8319} C_DIS
LIN {X 67.0393,Y -28.6521,Z 77,A -26.9914,B 24.8962,C -2.3515,E1 25.1488,E2 471.2761} C_DIS
LIN {X 68.6442,Y -24.561,Z 77,A -23.5531,B 24.8954,C -2.3616,E1 25.152,E2 467.8333} C_DIS
LIN {X 69.996,Y -20.3903,Z 77,A -21.5925,B 24.8983,C -2.3283,E1 25.1536,E2 465.9623} C_DIS
LIN {X 71.0532,Y -16.3253,Z 77,A -18.4088,B 24.8977,C -2.3352,E1 25.1558,E2 462.7807} C_DIS
LIN {X 71.5428,Y -14.0273,Z 77,A -16.4523,B 24.8969,C -2.3442,E1 25.1569,E2 460.8144} C_DIS
LIN {X 71.8833,Y -12.1604,Z 77,A -14.6057,B 24.8955,C -2.3594,E1 25.1578,E2 458.9427} C_DIS
LIN {X 72.67,Y -5.8437,Z 77,A -10.1591,B 24.8955,C -2.3589,E1 25.1593,E2 454.5236} C_DIS
LIN {X 72.8652,Y -2.4011,Z 77,A -6.4617,B 24.8922,C -2.3966,E1 25.1598,E2 450.7591} C_DIS
LIN {X 72.842,Y 3.0218,Z 77,A -2.5349,B 24.8919,C -2.4002,E1 25.1595,E2 446.8473} C_DIS
LIN {X 72.5861,Y 6.8074,Z 77,A 0.4565,B 24.891,C -2.4098,E1 25.1589,E2 443.8508} C_DIS
LIN {X 72.2007,Y 10.1072,Z 77,A 3.2175,B 24.8899,C -2.4224,E1 25.1578,E2 441.0764} C_DIS
LIN {X 71.4246,Y 14.615,Z 77,A 6.4158,B 24.8899,C -2.4218,E1 25.1562,E2 437.8982} C_DIS
LIN {X 70.3716,Y 19.05,Z 77,A 9.7554,B 24.8896,C -2.4256,E1 25.154,E2 434.5689} C_DIS
LIN {X 69.386,Y 22.3755,Z 77,A 13.013,B 24.8874,C -2.4492,E1 25.1513,E2 431.2742} C_DIS
LIN {X 68.1874,Y 25.7981,Z 77,A 15.5576,B 24.8874,C -2.4486,E1 25.1488,E2 428.7453} C_DIS
LIN {X 66.8132,Y 29.1731,Z 77,A 19.1113,B 24.8849,C -2.4768,E1 25.1449,E2 425.1443} C_DIS
LIN {X 65.317,Y 32.3845,Z 77,A 21.0101,B 24.8865,C -2.4588,E1 25.1426,E2 423.2982} C_DIS
LIN {X 63.8622,Y 35.1691,Z 77,A 23.8057,B 24.885,C -2.4748,E1 25.1389,E2 420.4794} C_DIS
LIN {X 61.7632,Y 38.7349,Z 77,A 26.5659,B 24.8856,C -2.4692,E1 25.135,E2 417.7465} C_DIS
LIN {X 60.4772,Y 40.7139,Z 77,A 28.9819,B 24.8836,C -2.49,E1 25.1312,E2 415.2934} C_DIS
LIN {X 57.9783,Y 44.2005,Z 77,A 32.2275,B 24.8832,C -2.4946,E1 25.1258,E2 412.0526} C_DIS
LIN {X 55.965,Y 46.7228,Z 77,A 34.395,B 24.8836,C -2.49,E1 25.122,E2 409.906} C_DIS
LIN {X 53.7254,Y 49.2814,Z 77,A 37.0945,B 24.883,C -2.4967,E1 25.117,E2 407.2026} C_DIS
LIN {X 52.0973,Y 51.0005,Z 77,A 39.102,B 24.8822,C -2.5048,E1 25.113,E2 405.1845} C_DIS
LIN {X 49.1935,Y 53.806,Z 77,A 42.3336,B 24.8815,C -2.5129,E1 25.1065,E2 401.947} C_DIS
LIN {X 46.3094,Y 56.3077,Z 77,A 45.1281,B 24.8815,C -2.5129,E1 25.1005,E2 399.1635} C_DIS
LIN {X 44.2316,Y 57.9542,Z 77,A 47.4775,B 24.8804,C -2.524,E1 25.0953,E2 396.7965} C_DIS
LIN {X 41.4483,Y 59.9762,Z 77,A 49.775,B 24.8811,C -2.5173,E1 25.0901,E2 394.5228} C_DIS
LIN {X 39.1318,Y 61.5131,Z 77,A 52.4321,B 24.8795,C -2.5337,E1 25.0838,E2 391.8355} C_DIS
LIN {X 35.3513,Y 63.7605,Z 77,A 56.0161,B 24.8787,C -2.542,E1 25.0751,E2 388.2425} C_DIS
LIN {X 31.6045,Y 65.698,Z 77,A 59.67,B 24.8774,C -2.5554,E1 25.0659,E2 384.5666} C_DIS
LIN {X 28.32,Y 67.1792,Z 77,A 61.8694,B 24.8788,C -2.5412,E1 25.0604,E2 382.4062} C_DIS
LIN {X 25.4982,Y 68.301,Z 77,A 64.126,B 24.8788,C -2.5399,E1 25.0545,E2 380.1574} C_DIS
LIN {X 22.5799,Y 69.3198,Z 77,A 67.4552,B 24.8764,C -2.5661,E1 25.0455,E2 376.7723} C_DIS
LIN {X 18.7085,Y 70.4639,Z 77,A 69.6092,B 24.8788,C -2.5409,E1 25.0399,E2 374.6818} C_DIS
LIN {X 16.787,Y 70.9466,Z 77,A 72.1159,B 24.8763,C -2.567,E1 25.0329,E2 372.1166} C_DIS
LIN {X 13.0548,Y 71.7263,Z 77,A 73.8009,B 24.8795,C -2.5336,E1 25.0285,E2 370.513} C_DIS
LIN {X 8.1628,Y 72.4468,Z 77,A 77.6278,B 24.8795,C -2.533,E1 25.018,E2 366.6909} C_DIS
LIN {X 3.4297,Y 72.8244,Z 77,A 81.5261,B 24.8791,C -2.5374,E1 25.0071,E2 362.7841} C_DIS
LIN {X -1.2156,Y 72.8945,Z 77,A 85.3057,B 24.8789,C -2.54,E1 24.9965,E2 358.9985} C_DIS
LIN {X -4.8412,Y 72.7436,Z 77,A 88.6646,B 24.8777,C -2.5519,E1 24.9871,E2 355.6104} C_DIS
LIN {X -7.6653,Y 72.5005,Z 77,A 91.0411,B 24.8775,C -2.5545,E1 24.9804,E2 353.2263} C_DIS
LIN {X -13.1784,Y 71.7041,Z 77,A 94.903,B 24.879,C -2.5385,E1 24.9699,E2 349.3992} C_DIS
LIN {X -16.6302,Y 70.9828,Z 77,A 97.9506,B 24.8786,C -2.543,E1 24.9615,E2 346.3371} C_DIS
LIN {X -20.5775,Y 69.9404,Z 77,A 100.5413,B 24.8804,C -2.5244,E1 24.9547,E2 343.7865} C_DIS
LIN {X -22.2332,Y 69.432,Z 77,A 103.1194,B 24.8777,C -2.5529,E1 24.9476,E2 341.136} C_DIS
LIN {X -25.6285,Y 68.2517,Z 77,A 104.9474,B 24.8803,C -2.5247,E1 24.943,E2 339.3714} C_DIS
LIN {X -30.0426,Y 66.4268,Z 77,A 108.6411,B 24.881,C -2.5179,E1 24.9335,E2 335.6854} C_DIS
LIN {X -33.2042,Y 64.9042,Z 77,A 111.9395,B 24.8802,C -2.5266,E1 24.9252,E2 332.3575} C_DIS
LIN {X -37.2515,Y 62.6692,Z 77,A 114.9233,B 24.8822,C -2.5047,E1 24.918,E2 329.4172} C_DIS
LIN {X -40.0706,Y 60.905,Z 77,A 117.9184,B 24.8818,C -2.509,E1 24.9109,E2 326.4025} C_DIS
LIN {X -42.3885,Y 59.3152,Z 77,A 120.648,B 24.8811,C -2.517,E1 24.9046,E2 323.6443} C_DIS
LIN {X -46.1765,Y 56.4174,Z 77,A 123.6319,B 24.8835,C -2.4909,E1 24.8982,E2 320.7116} C_DIS
LIN {X -48.2786,Y 54.6299,Z 77,A 126.4584,B 24.8825,C -2.5016,E1 24.8921,E2 317.8486} C_DIS
LIN {X -50.7723,Y 52.3193,Z 77,A 129.1026,B 24.8832,C -2.4947,E1 24.8868,E2 315.2098} C_DIS
LIN {X -53.7883,Y 49.2128,Z 77,A 132.2555,B 24.8845,C -2.4806,E1 24.8808,E2 312.0769} C_DIS
LIN {X -55.5632,Y 47.1997,Z 77,A 134.4328,B 24.8849,C -2.4768,E1 24.8768,E2 309.8987} C_DIS
LIN {X -57.5437,Y 44.765,Z 77,A 137.164,B 24.8849,C -2.4765,E1 24.8721,E2 307.1554} C_DIS
LIN {X -60.3881,Y 40.8455,Z 77,A 140.5958,B 24.8866,C -2.4576,E1 24.8666,E2 303.7521} C_DIS
LIN {X -62.0225,Y 38.3199,Z 77,A 143.1007,B 24.887,C -2.4542,E1 24.8629,E2 301.2425} C_DIS
LIN {X -64.5456,Y 33.896,Z 77,A 146.9,B 24.8884,C -2.4381,E1 24.8577,E2 297.4617} C_DIS
LIN {X -65.9313,Y 31.1151,Z 77,A 149.8949,B 24.8879,C -2.4436,E1 24.854,E2 294.4375} C_DIS
LIN {X -67.6316,Y 27.2234,Z 77,A 152.9531,B 24.8894,C -2.4271,E1 24.8507,E2 291.4016} C_DIS
LIN {X -68.5243,Y 24.8897,Z 77,A 154.6376,B 24.8906,C -2.4148,E1 24.8491,E2 289.737} C_DIS
LIN {X -69.1742,Y 23.0234,Z 77,A 156.2444,B 24.8909,C -2.4113,E1 24.8477,E2 288.1295} C_DIS
LIN {X -69.9219,Y 20.6399,Z 77,A 159.2308,B 24.8893,C -2.4286,E1 24.8453,E2 285.0845} C_DIS
LIN {X -70.8667,Y 17.1176,Z 77,A 161.0731,B 24.8922,C -2.3962,E1 24.8441,E2 283.3088} C_DIS
LIN {X -71.261,Y 15.3928,Z 77,A 163.0747,B 24.8914,C -2.4058,E1 24.8429,E2 281.2727} C_DIS
LIN {X -71.9341,Y 11.8565,Z 77,A 165.3997,B 24.8932,C -2.3854,E1 24.8417,E2 278.9826} C_DIS
LIN {X -72.3628,Y 8.8801,Z 77,A 168.1246,B 24.8932,C -2.3861,E1 24.8407,E2 276.2398} C_DIS
LIN {X -72.7517,Y 4.7225,Z 77,A 171.1881,B 24.8945,C -2.3707,E1 24.84,E2 273.1946} C_DIS
LIN {X -72.8886,Y 1.5342,Z 77,A 173.8637,B 24.8949,C -2.3665,E1 24.8398,E2 270.5128} C_DIS
LIN {X -72.8889,Y -1.5211,Z 77,A 176.1876,B 24.8957,C -2.3572,E1 24.8398,E2 268.1972} C_DIS
LIN {X -72.7454,Y -4.8157,Z 77,A 179.0059,B 24.896,C -2.3542,E1 24.8403,E2 265.3692} C_DIS
LIN {X -72.4873,Y -7.7907,Z 77,A -178.8293,B 24.897,C -2.3426,E1 24.8409,E2 263.2189} C_DIS
LIN {X -71.9335,Y -11.8602,Z 77,A -175.0592,B 24.8968,C -2.3451,E1 24.8425,E2 259.4206} C_DIS
LIN {X -71.1521,Y -15.8926,Z 77,A -172.1984,B 24.8984,C -2.3267,E1 24.8441,E2 256.5868} C_DIS
LIN {X -69.7268,Y -21.2919,Z 77,A -167.94,B 24.8998,C -2.3105,E1 24.8473,E2 252.3423} C_DIS
LIN {X -68.821,Y -24.0572,Z 77,A -164.7855,B 24.8987,C -2.324,E1 24.8502,E2 249.1377} C_DIS
LIN {X -67.5136,Y -27.5133,Z 77,A -162.8065,B 24.9013,C -2.2941,E1 24.8522,E2 247.219} C_DIS
LIN {X -65.7614,Y -31.4725,Z 77,A -159.7306,B 24.9027,C -2.277,E1 24.8557,E2 244.167} C_DIS
LIN {X -64.5197,Y -33.9452,Z 77,A -156.5994,B 24.9013,C -2.2934,E1 24.8598,E2 240.9801} C_DIS
LIN {X -62.8151,Y -37.0046,Z 77,A -154.3315,B 24.9029,C -2.2747,E1 24.8629,E2 238.7448} C_DIS
LIN {X -60.0881,Y -41.2868,Z 77,A -150.6004,B 24.9043,C -2.2585,E1 24.8685,E2 235.0337} C_DIS
LIN {X -57.8139,Y -44.4143,Z 77,A -147.491,B 24.9048,C -2.2528,E1 24.8737,E2 231.9229} C_DIS
LIN {X -55.5023,Y -47.2712,Z 77,A -144.4702,B 24.9051,C -2.2492,E1 24.879,E2 228.8966} C_DIS
LIN {X -53.7755,Y -49.2268,Z 77,A -142.369,B 24.9054,C -2.2459,E1 24.8829,E2 226.7939} C_DIS
LIN {X -50.5662,Y -52.5179,Z 77,A -138.8177,B 24.9061,C -2.2368,E1 24.8899,E2 223.2492} C_DIS
LIN {X -47.5127,Y -55.2965,Z 77,A -135.7057,B 24.9069,C -2.2272,E1 24.8964,E2 220.1475} C_DIS
LIN {X -45.2579,Y -57.1559,Z 77,A -133.5613,B 24.9076,C -2.2193,E1 24.901,E2 218.0139} C_DIS
LIN {X -43.5246,Y -58.4875,Z 77,A -131.3265,B 24.9068,C -2.2289,E1 24.906,E2 215.7482} C_DIS
LIN {X -41.1976,Y -60.1497,Z 77,A -129.0914,B 24.9071,C -2.2249,E1 24.9111,E2 213.5149} C_DIS
LIN {X -37.7715,Y -62.357,Z 77,A -125.3777,B 24.9065,C -2.2328,E1 24.92,E2 209.7707} C_DIS
LIN {X -34.8482,Y -64.0365,Z 77,A -122.3168,B 24.9059,C -2.2397,E1 24.9276,E2 206.6849} C_DIS
LIN {X -31.3352,Y -65.8274,Z 77,A -119.9882,B 24.9078,C -2.2165,E1 24.9333,E2 204.4053} C_DIS
LIN {X -28.7538,Y -66.996,Z 77,A -117.8114,B 24.9081,C -2.2129,E1 24.9388,E2 202.232} C_DIS
LIN {X -25.9652,Y -68.1242,Z 77,A -114.3413,B 24.906,C -2.239,E1 24.9481,E2 198.6925} C_DIS
LIN {X -21.5797,Y -69.6374,Z 77,A -112.0311,B 24.9091,C -2.2019,E1 24.954,E2 196.4663} C_DIS
LIN {X -19.8787,Y -70.142,Z 77,A -109.4843,B 24.9067,C -2.2307,E1 24.9611,E2 193.847} C_DIS
LIN {X -15.8503,Y -71.1614,Z 77,A -107.39,B 24.9093,C -2.1987,E1 24.9665,E2 191.826} C_DIS
LIN {X -12.1257,Y -71.8891,Z 77,A -104.369,B 24.9093,C -2.1987,E1 24.9748,E2 188.8021} C_DIS
LIN {X -6.768,Y -72.5897,Z 77,A -100.379,B 24.9099,C -2.1912,E1 24.9859,E2 184.8269} C_DIS
LIN {X -1.9795,Y -72.8781,Z 77,A -96.7126,B 24.9102,C -2.1886,E1 24.9961,E2 181.1655} C_DIS
LIN {X 0.4854,Y -72.8916,Z 77,A -95.3086,B 24.9113,C -2.1752,E1 24.9999,E2 179.7932} C_DIS
Enddeposition()
LIN {X 0.4854,Y -72.8916,Z 77,A -95.3086,B 24.9113,C -2.1752,E1 24.9999,E2 179.7932} C_DIS
Startdeposition()
$VEL.CP = VEL_PRINT
LIN {X -0.8385,Y -71.9485,Z 77,A -96.2201,B 24.9096,C -2.1951,E1 24.9975,E2 180.6574} C_DIS
LIN {X -5.9619,Y -71.7052,Z 77,A -100.1824,B 24.9094,C -2.198,E1 24.9865,E2 184.614} C_DIS
LIN {X -10.3838,Y -71.1996,Z 77,A -103.8582,B 24.9096,C -2.1952,E1 24.9762,E2 188.299} C_DIS
LIN {X -13.5156,Y -70.6716,Z 77,A -106.7707,B 24.9103,C -2.1864,E1 24.9681,E2 191.2353} C_DIS
LIN {X -16.8471,Y -69.9518,Z 77,A -109.5588,B 24.9103,C -2.1859,E1 24.9605,E2 194.0283} C_DIS
LIN {X -20.3526,Y -69.0139,Z 77,A -112.5113,B 24.9103,C -2.1862,E1 24.9526,E2 196.9847} C_DIS
LIN {X -25.7552,Y -67.1855,Z 77,A -116.7887,B 24.9095,C -2.1965,E1 24.9414,E2 201.246} C_DIS
LIN {X -28.4422,Y -66.093,Z 77,A -119.4558,B 24.91,C -2.1902,E1 24.9345,E2 203.9342} C_DIS
LIN {X -32.9363,Y -63.9716,Z 77,A -123.0993,B 24.909,C -2.2025,E1 24.9254,E2 207.5581} C_DIS
LIN {X -35.9048,Y -62.3534,Z 77,A -126.9225,B 24.9109,C -2.1795,E1 24.916,E2 211.4472} C_DIS
LIN {X -39.82,Y -59.9297,Z 77,A -129.4942,B 24.9083,C -2.2108,E1 24.9101,E2 213.9527} C_DIS
LIN {X -42.5089,Y -58.0528,Z 77,A -132.1534,B 24.9081,C -2.214,E1 24.904,E2 216.6135} C_DIS
LIN {X -45.9009,Y -55.4098,Z 77,A -135.3858,B 24.9072,C -2.2247,E1 24.897,E2 219.8325} C_DIS
LIN {X -49.2967,Y -52.4115,Z 77,A -139.0335,B 24.9067,C -2.2308,E1 24.8894,E2 223.4803} C_DIS
LIN {X -52.2123,Y -49.5086,Z 77,A -142.3912,B 24.9062,C -2.2357,E1 24.8828,E2 226.8404} C_DIS
Enddeposition()
END
